(* LS Electric XG5000 project: 201209_AX_ROOF *)
(* PLC NewPLC *)
(* module base 0 slot 0: FEnet:XGL-EFMT(B) (Fast Ethernet 통신 모듈, 전기 Master) *)
(* module base 0 slot 1: FEnet:XGL-EFMT(B) (Fast Ethernet 통신 모듈, 전기 Master) *)
(* module base 0 slot 2: FEnet:XGL-EFMT(B) (Fast Ethernet 통신 모듈, 전기 Master) *)
(* module base 0 slot 3: FEnet:XGL-EFMT(B) (Fast Ethernet 통신 모듈, 전기 Master) *)
(* module base 0 slot 4: FEnet:XGL-EFMT(B) (Fast Ethernet 통신 모듈, 전기 Master) *)
(* module base 0 slot 5: FEnet:XGL-EFMT(B) (Fast Ethernet 통신 모듈, 전기 Master) *)
(* module base 0 slot 6: FEnet:XGL-EFMT(B) (Fast Ethernet 통신 모듈, 전기 Master) *)
(* module base 0 slot 7: FEnet:XGL-EFMT(B) (Fast Ethernet 통신 모듈, 전기 Master) *)
(* module base 0 slot 8: Pnet:XGL-PMEC/B (Pnet 통신 모듈, Profibus-DP Master) *)
(* module base 0 slot 0: 입력 모듈:XBE-DC16A/B (DC24V 입력, 16점 / DC12/24V 입력, 16점) *)
(* module base 0 slot 1: 입력 모듈:XBE-DC16A/B (DC24V 입력, 16점 / DC12/24V 입력, 16점) *)
(* module base 0 slot 2: 입력 모듈:XBE-DC16A/B (DC24V 입력, 16점 / DC12/24V 입력, 16점) *)
(* module base 0 slot 3: 입력 모듈:XBE-DC16A/B (DC24V 입력, 16점 / DC12/24V 입력, 16점) *)
(* module base 0 slot 4: 출력 모듈:XBE-TN/TP16A (트랜지스터 출력, 16점 (싱크출력/소스출력)) *)
(* module base 0 slot 5: 출력 모듈:XBE-TN/TP16A (트랜지스터 출력, 16점 (싱크출력/소스출력)) *)
(* module base 0 slot 6: 출력 모듈:XBE-TN/TP16A (트랜지스터 출력, 16점 (싱크출력/소스출력)) *)
(* module base 0 slot 7: 출력 모듈:XBE-TN/TP16A (트랜지스터 출력, 16점 (싱크출력/소스출력)) *)
(* module base 0 slot 0: 입력 모듈:XBE-DC16A/B (DC24V 입력, 16점 / DC12/24V 입력, 16점) *)
(* module base 0 slot 1: 입력 모듈:XBE-DC16A/B (DC24V 입력, 16점 / DC12/24V 입력, 16점) *)
(* module base 0 slot 2: 입력 모듈:XBE-DC16A/B (DC24V 입력, 16점 / DC12/24V 입력, 16점) *)
(* module base 0 slot 3: 입력 모듈:XBE-DC16A/B (DC24V 입력, 16점 / DC12/24V 입력, 16점) *)
(* module base 0 slot 4: 출력 모듈:XBE-TN/TP16A (트랜지스터 출력, 16점 (싱크출력/소스출력)) *)
(* module base 0 slot 5: 출력 모듈:XBE-TN/TP16A (트랜지스터 출력, 16점 (싱크출력/소스출력)) *)
(* module base 0 slot 6: 출력 모듈:XBE-TN/TP16A (트랜지스터 출력, 16점 (싱크출력/소스출력)) *)
(* module base 0 slot 7: 출력 모듈:XBE-TN/TP16A (트랜지스터 출력, 16점 (싱크출력/소스출력)) *)
(* module base 0 slot 0: 입력 모듈:XBE-DC16A/B (DC24V 입력, 16점 / DC12/24V 입력, 16점) *)
(* module base 0 slot 1: 입력 모듈:XBE-DC16A/B (DC24V 입력, 16점 / DC12/24V 입력, 16점) *)
(* module base 0 slot 2: 입력 모듈:XBE-DC16A/B (DC24V 입력, 16점 / DC12/24V 입력, 16점) *)
(* module base 0 slot 3: 출력 모듈:XBE-TN/TP16A (트랜지스터 출력, 16점 (싱크출력/소스출력)) *)
(* module base 0 slot 4: 출력 모듈:XBE-TN/TP16A (트랜지스터 출력, 16점 (싱크출력/소스출력)) *)
(* module base 0 slot 0: 입력 모듈:XBE-DC16A/B (DC24V 입력, 16점 / DC12/24V 입력, 16점) *)
(* module base 0 slot 1: 입력 모듈:XBE-DC16A/B (DC24V 입력, 16점 / DC12/24V 입력, 16점) *)
(* module base 0 slot 2: 입력 모듈:XBE-DC16A/B (DC24V 입력, 16점 / DC12/24V 입력, 16점) *)
(* module base 0 slot 3: 출력 모듈:XBE-TN/TP16A (트랜지스터 출력, 16점 (싱크출력/소스출력)) *)
(* module base 0 slot 4: 출력 모듈:XBE-TN/TP16A (트랜지스터 출력, 16점 (싱크출력/소스출력)) *)
(* module base 0 slot 0: 입력 모듈:XBE-DC16A/B (DC24V 입력, 16점 / DC12/24V 입력, 16점) *)
(* module base 0 slot 1: 입력 모듈:XBE-DC16A/B (DC24V 입력, 16점 / DC12/24V 입력, 16점) *)
(* module base 0 slot 2: 입력 모듈:XBE-DC16A/B (DC24V 입력, 16점 / DC12/24V 입력, 16점) *)
(* module base 0 slot 3: 출력 모듈:XBE-TN/TP16A (트랜지스터 출력, 16점 (싱크출력/소스출력)) *)
(* module base 0 slot 4: 출력 모듈:XBE-TN/TP16A (트랜지스터 출력, 16점 (싱크출력/소스출력)) *)
(* module base 0 slot 0: 입력 모듈:XBE-DC16A/B (DC24V 입력, 16점 / DC12/24V 입력, 16점) *)
(* module base 0 slot 1: 입력 모듈:XBE-DC16A/B (DC24V 입력, 16점 / DC12/24V 입력, 16점) *)
(* module base 0 slot 2: 입력 모듈:XBE-DC16A/B (DC24V 입력, 16점 / DC12/24V 입력, 16점) *)
(* module base 0 slot 3: 출력 모듈:XBE-TN/TP16A (트랜지스터 출력, 16점 (싱크출력/소스출력)) *)
(* module base 0 slot 4: 출력 모듈:XBE-TN/TP16A (트랜지스터 출력, 16점 (싱크출력/소스출력)) *)
(* module base 0 slot 0: 입력 모듈:XBE-DC16A/B (DC24V 입력, 16점 / DC12/24V 입력, 16점) *)
(* module base 0 slot 1: 입력 모듈:XBE-DC16A/B (DC24V 입력, 16점 / DC12/24V 입력, 16점) *)
(* module base 0 slot 2: 입력 모듈:XBE-DC16A/B (DC24V 입력, 16점 / DC12/24V 입력, 16점) *)
(* module base 0 slot 3: 출력 모듈:XBE-TN/TP16A (트랜지스터 출력, 16점 (싱크출력/소스출력)) *)
(* module base 0 slot 4: 출력 모듈:XBE-TN/TP16A (트랜지스터 출력, 16점 (싱크출력/소스출력)) *)
(* module base 0 slot 0: 입력 모듈:XBE-DC16A/B (DC24V 입력, 16점 / DC12/24V 입력, 16점) *)
(* module base 0 slot 1: 입력 모듈:XBE-DC16A/B (DC24V 입력, 16점 / DC12/24V 입력, 16점) *)
(* module base 0 slot 2: 입력 모듈:XBE-DC16A/B (DC24V 입력, 16점 / DC12/24V 입력, 16점) *)
(* module base 0 slot 3: 출력 모듈:XBE-TN/TP16A (트랜지스터 출력, 16점 (싱크출력/소스출력)) *)
(* module base 0 slot 4: 출력 모듈:XBE-TN/TP16A (트랜지스터 출력, 16점 (싱크출력/소스출력)) *)
(* module base 0 slot 0: 입력 모듈:XBE-DC16A/B (DC24V 입력, 16점 / DC12/24V 입력, 16점) *)
(* module base 0 slot 1: 입력 모듈:XBE-DC16A/B (DC24V 입력, 16점 / DC12/24V 입력, 16점) *)
(* module base 0 slot 2: 입력 모듈:XBE-DC16A/B (DC24V 입력, 16점 / DC12/24V 입력, 16점) *)
(* module base 0 slot 3: 출력 모듈:XBE-TN/TP16A (트랜지스터 출력, 16점 (싱크출력/소스출력)) *)
(* module base 0 slot 4: 출력 모듈:XBE-TN/TP16A (트랜지스터 출력, 16점 (싱크출력/소스출력)) *)
(* module base 0 slot 0: 입력 모듈:XBE-DC16A/B (DC24V 입력, 16점 / DC12/24V 입력, 16점) *)
(* module base 0 slot 1: 입력 모듈:XBE-DC16A/B (DC24V 입력, 16점 / DC12/24V 입력, 16점) *)
(* module base 0 slot 2: 입력 모듈:XBE-DC16A/B (DC24V 입력, 16점 / DC12/24V 입력, 16점) *)
(* module base 0 slot 3: 출력 모듈:XBE-TN/TP16A (트랜지스터 출력, 16점 (싱크출력/소스출력)) *)
(* module base 0 slot 4: 출력 모듈:XBE-TN/TP16A (트랜지스터 출력, 16점 (싱크출력/소스출력)) *)
(* module base 0 slot 0: 입력 모듈:XBE-DC16A/B (DC24V 입력, 16점 / DC12/24V 입력, 16점) *)
(* module base 0 slot 1: 입력 모듈:XBE-DC16A/B (DC24V 입력, 16점 / DC12/24V 입력, 16점) *)
(* module base 0 slot 2: 입력 모듈:XBE-DC16A/B (DC24V 입력, 16점 / DC12/24V 입력, 16점) *)
(* module base 0 slot 3: 출력 모듈:XBE-TN/TP16A (트랜지스터 출력, 16점 (싱크출력/소스출력)) *)
(* module base 0 slot 4: 출력 모듈:XBE-TN/TP16A (트랜지스터 출력, 16점 (싱크출력/소스출력)) *)
(* module base 0 slot 0: 입력 모듈:XBE-DC16A/B (DC24V 입력, 16점 / DC12/24V 입력, 16점) *)
(* module base 0 slot 1: 출력 모듈:XBE-TN/TP16A (트랜지스터 출력, 16점 (싱크출력/소스출력)) *)
(* module base 0 slot 2: 입력 모듈:XBE-DC16A/B (DC24V 입력, 16점 / DC12/24V 입력, 16점) *)
(* module base 0 slot 3: 출력 모듈:XBE-TN/TP16A (트랜지스터 출력, 16점 (싱크출력/소스출력)) *)
(* module base 0 slot 0: 입력 모듈:XBE-DC16A/B (DC24V 입력, 16점 / DC12/24V 입력, 16점) *)
(* module base 0 slot 1: 출력 모듈:XBE-TN/TP16A (트랜지스터 출력, 16점 (싱크출력/소스출력)) *)
(* module base 0 slot 2: 입력 모듈:XBE-DC16A/B (DC24V 입력, 16점 / DC12/24V 입력, 16점) *)
(* module base 0 slot 3: 출력 모듈:XBE-TN/TP16A (트랜지스터 출력, 16점 (싱크출력/소스출력)) *)
(* module base 0 slot 0: 입력 모듈:XBE-DC16A/B (DC24V 입력, 16점 / DC12/24V 입력, 16점) *)
(* module base 0 slot 1: 출력 모듈:XBE-TN/TP16A (트랜지스터 출력, 16점 (싱크출력/소스출력)) *)
(* module base 0 slot 2: 입력 모듈:XBE-DC16A/B (DC24V 입력, 16점 / DC12/24V 입력, 16점) *)
(* module base 0 slot 3: 출력 모듈:XBE-TN/TP16A (트랜지스터 출력, 16점 (싱크출력/소스출력)) *)
(* module base 0 slot 0: 입력 모듈:XBE-DC16A/B (DC24V 입력, 16점 / DC12/24V 입력, 16점) *)
(* module base 0 slot 1: 입력 모듈:XBE-DC16A/B (DC24V 입력, 16점 / DC12/24V 입력, 16점) *)
(* module base 0 slot 2: 입력 모듈:XBE-DC16A/B (DC24V 입력, 16점 / DC12/24V 입력, 16점) *)
(* module base 0 slot 3: 출력 모듈:XBE-TN/TP16A (트랜지스터 출력, 16점 (싱크출력/소스출력)) *)
(* module base 0 slot 4: 출력 모듈:XBE-TN/TP16A (트랜지스터 출력, 16점 (싱크출력/소스출력)) *)
(* module base 0 slot 5: 입력 모듈:XBE-DC16A/B (DC24V 입력, 16점 / DC12/24V 입력, 16점) *)
(* module base 0 slot 6: 출력 모듈:XBE-TN/TP16A (트랜지스터 출력, 16점 (싱크출력/소스출력)) *)
(* module base 0 slot 0: 입력 모듈:XBE-DC16A/B (DC24V 입력, 16점 / DC12/24V 입력, 16점) *)
(* module base 0 slot 1: 출력 모듈:XBE-TN/TP16A (트랜지스터 출력, 16점 (싱크출력/소스출력)) *)
(* module base 0 slot 2: 입력 모듈:XBE-DC16A/B (DC24V 입력, 16점 / DC12/24V 입력, 16점) *)
(* module base 0 slot 3: 출력 모듈:XBE-TN/TP16A (트랜지스터 출력, 16점 (싱크출력/소스출력)) *)
(* module base 0 slot 0: 입력 모듈:XBE-DC16A/B (DC24V 입력, 16점 / DC12/24V 입력, 16점) *)
(* module base 0 slot 1: 출력 모듈:XBE-TN/TP16A (트랜지스터 출력, 16점 (싱크출력/소스출력)) *)
(* module base 0 slot 2: 입력 모듈:XBE-DC16A/B (DC24V 입력, 16점 / DC12/24V 입력, 16점) *)
(* module base 0 slot 3: 출력 모듈:XBE-TN/TP16A (트랜지스터 출력, 16점 (싱크출력/소스출력)) *)
(* module base 0 slot 0: 입력 모듈:XBE-DC16A/B (DC24V 입력, 16점 / DC12/24V 입력, 16점) *)
(* module base 0 slot 1: 입력 모듈:XBE-DC16A/B (DC24V 입력, 16점 / DC12/24V 입력, 16점) *)
(* module base 0 slot 2: 입력 모듈:XBE-DC16A/B (DC24V 입력, 16점 / DC12/24V 입력, 16점) *)
(* module base 0 slot 3: 출력 모듈:XBE-TN/TP16A (트랜지스터 출력, 16점 (싱크출력/소스출력)) *)
(* module base 0 slot 4: 출력 모듈:XBE-TN/TP16A (트랜지스터 출력, 16점 (싱크출력/소스출력)) *)
(* module base 0 slot 5: 입력 모듈:XBE-DC16A/B (DC24V 입력, 16점 / DC12/24V 입력, 16점) *)
(* module base 0 slot 6: 출력 모듈:XBE-TN/TP16A (트랜지스터 출력, 16점 (싱크출력/소스출력)) *)
(* module base 0 slot 0: 입력 모듈:XBE-DC16A/B (DC24V 입력, 16점 / DC12/24V 입력, 16점) *)
(* module base 0 slot 1: 입력 모듈:XBE-DC16A/B (DC24V 입력, 16점 / DC12/24V 입력, 16점) *)
(* module base 0 slot 2: 입력 모듈:XBE-DC16A/B (DC24V 입력, 16점 / DC12/24V 입력, 16점) *)
(* module base 0 slot 3: 출력 모듈:XBE-TN/TP16A (트랜지스터 출력, 16점 (싱크출력/소스출력)) *)
(* module base 0 slot 4: 출력 모듈:XBE-TN/TP16A (트랜지스터 출력, 16점 (싱크출력/소스출력)) *)
(* module base 0 slot 5: 입력 모듈:XBE-DC16A/B (DC24V 입력, 16점 / DC12/24V 입력, 16점) *)
(* module base 0 slot 6: 출력 모듈:XBE-TN/TP16A (트랜지스터 출력, 16점 (싱크출력/소스출력)) *)
(* module base 0 slot 0: 입력 모듈:XBE-DC16A/B (DC24V 입력, 16점 / DC12/24V 입력, 16점) *)
(* module base 0 slot 1: 입력 모듈:XBE-DC16A/B (DC24V 입력, 16점 / DC12/24V 입력, 16점) *)
(* module base 0 slot 2: 출력 모듈:XBE-TN/TP16A (트랜지스터 출력, 16점 (싱크출력/소스출력)) *)
(* module base 0 slot 3: 입력 모듈:XBE-DC16A/B (DC24V 입력, 16점 / DC12/24V 입력, 16점) *)
(* module base 0 slot 4: 출력 모듈:XBE-TN/TP16A (트랜지스터 출력, 16점 (싱크출력/소스출력)) *)
(* module base 0 slot 0: 입력 모듈:XBE-DC16A/B (DC24V 입력, 16점 / DC12/24V 입력, 16점) *)
(* module base 0 slot 1: 입력 모듈:XBE-DC16A/B (DC24V 입력, 16점 / DC12/24V 입력, 16점) *)
(* module base 0 slot 2: 출력 모듈:XBE-TN/TP16A (트랜지스터 출력, 16점 (싱크출력/소스출력)) *)
(* module base 0 slot 3: 입력 모듈:XBE-DC16A/B (DC24V 입력, 16점 / DC12/24V 입력, 16점) *)
(* module base 0 slot 4: 출력 모듈:XBE-TN/TP16A (트랜지스터 출력, 16점 (싱크출력/소스출력)) *)
(* module base 0 slot 0: 입력 모듈:XBE-DC16A/B (DC24V 입력, 16점 / DC12/24V 입력, 16점) *)
(* module base 0 slot 1: 입력 모듈:XBE-DC16A/B (DC24V 입력, 16점 / DC12/24V 입력, 16점) *)
(* module base 0 slot 2: 출력 모듈:XBE-TN/TP16A (트랜지스터 출력, 16점 (싱크출력/소스출력)) *)
(* module base 0 slot 3: 입력 모듈:XBE-DC16A/B (DC24V 입력, 16점 / DC12/24V 입력, 16점) *)
(* module base 0 slot 4: 출력 모듈:XBE-TN/TP16A (트랜지스터 출력, 16점 (싱크출력/소스출력)) *)
(* module base 0 slot 0: 입력 모듈:XBE-DC16A/B (DC24V 입력, 16점 / DC12/24V 입력, 16점) *)
(* module base 0 slot 1: 입력 모듈:XBE-DC16A/B (DC24V 입력, 16점 / DC12/24V 입력, 16점) *)
(* module base 0 slot 2: 입력 모듈:XBE-DC16A/B (DC24V 입력, 16점 / DC12/24V 입력, 16점) *)
(* module base 0 slot 3: 출력 모듈:XBE-TN/TP16A (트랜지스터 출력, 16점 (싱크출력/소스출력)) *)
(* module base 0 slot 4: 출력 모듈:XBE-TN/TP16A (트랜지스터 출력, 16점 (싱크출력/소스출력)) *)
(* module base 0 slot 5: 입력 모듈:XBE-DC16A/B (DC24V 입력, 16점 / DC12/24V 입력, 16점) *)
(* module base 0 slot 6: 출력 모듈:XBE-TN/TP16A (트랜지스터 출력, 16점 (싱크출력/소스출력)) *)
VAR_GLOBAL RETAIN
    ALWAYS_OFF AT %MW3.0 : BOOL; (* 항시 OFF *)
    ALWAYS_ON AT %MW3.1 : BOOL; (* 항시 ON *)
    CARTYPE AT %MW10000 : ARRAY[0..599] OF WORD; (* CARTYPE *)
    CLOCK_BIT_0_1Sec AT %MW0.0 : BOOL; (* CLOCK_BIT_0_1Sec *)
    CLOCK_BIT_0_2Sec AT %MW0.1 : BOOL; (* CLOCK_BIT_0_2Sec *)
    CLOCK_BIT_0_4Sec AT %MW0.2 : BOOL; (* CLOCK_BIT_0_4Sec *)
    CLOCK_BIT_0_5Sec AT %MW0.3 : BOOL; (* 플리커 0.5초 *)
    CLOCK_BIT_0_8Sec AT %MW0.4 : BOOL; (* CLOCK_BIT_0_8Sec *)
    CLOCK_BIT_1_0Sec AT %MW0.5 : BOOL; (* CLOCK_BIT_1_0Sec *)
    CLOCK_BIT_1_6Sec AT %MW0.6 : BOOL; (* CLOCK_BIT_1_6Sec *)
    CLOCK_BIT_2_0Sec AT %MW0.7 : BOOL; (* CLOCK_BIT_2_0Sec *)
    GATE1_M_CP_TRIP AT %MW400.15 : BOOL; (* GATEBOX1 CP OFF 이상 *)
    GATE1_M_EMSTOP AT %MW400.7 : BOOL; (* GATE1 비상정지 이상 *)
    GATE1_M_GATE_CLOSE AT %MW400.3 : BOOL; (* GATE1_M_GATE_CLOSE *)
    GATE1_M_GATE_OPEN AT %MW400.13 : BOOL; (* GATEBOX1 이상 *)
    GATE1_M_GATE_열림_보조 AT %MW400.12 : BOOL; (* GATE1_M_GATE_열림_보조 *)
    GATE1_M_RESTART AT %MW400.1 : BOOL; (* GATE1_M_RESTART *)
    GATE1_M_STOP_CALL AT %MW400.2 : BOOL; (* GATE1_M_STOP_CALL *)
    GATE1_M_비상정지_정상 AT %MW400.4 : BOOL;
    GATE1_M_이상_리셋 AT %MW400.0 : BOOL; (* GATE1 PB 이상리셋 *)
    GATE1_M_통신_이상 AT %MW400.14 : BOOL; (* GATEBOX1 통신이상 *)
    GATE2_M_CP_TRIP AT %MW401.15 : BOOL; (* GATEBOX2 CP OFF 이상 *)
    GATE2_M_EMSTOP AT %MW401.7 : BOOL; (* GATE2 비상정지 이상 *)
    GATE2_M_GATE_CLOSE AT %MW401.3 : BOOL; (* GATE2_M_GATE_CLOSE *)
    GATE2_M_GATE_OPEN AT %MW401.13 : BOOL; (* GATEBOX2 이상 *)
    GATE2_M_GATE_열림_보조 AT %MW401.12 : BOOL; (* GATE2_M_GATE_열림_보조 *)
    GATE2_M_RESTART AT %MW401.1 : BOOL; (* GATE2_M_RESTART *)
    GATE2_M_STOP_CALL AT %MW401.2 : BOOL; (* GATE2_M_STOP_CALL *)
    GATE2_M_비상정지_정상 AT %MW401.4 : BOOL;
    GATE2_M_이상_리셋 AT %MW401.0 : BOOL; (* GATE2 PB 이상리셋 *)
    GATE2_M_통신_이상 AT %MW401.14 : BOOL; (* GATEBOX2 통신이상 *)
    GATE3_M_CP_TRIP AT %MW402.15 : BOOL; (* GATEBOX3 CP OFF 이상 *)
    GATE3_M_EMSTOP AT %MW402.7 : BOOL; (* GATE3 비상정지 이상 *)
    GATE3_M_GATE_CLOSE AT %MW402.3 : BOOL; (* GATE3_M_GATE_CLOSE *)
    GATE3_M_GATE_OPEN AT %MW402.13 : BOOL; (* GATEBOX3 이상 *)
    GATE3_M_GATE_열림_보조 AT %MW402.12 : BOOL; (* GATE3_M_GATE_열림_보조 *)
    GATE3_M_RESTART AT %MW402.1 : BOOL; (* GATE3_M_RESTART *)
    GATE3_M_STOP_CALL AT %MW402.2 : BOOL; (* GATE3_M_STOP_CALL *)
    GATE3_M_비상정지_정상 AT %MW402.4 : BOOL;
    GATE3_M_이상_리셋 AT %MW402.0 : BOOL; (* GATE3 PB 이상리셋 *)
    GATE3_M_통신_이상 AT %MW402.14 : BOOL; (* GATEBOX3 통신이상 *)
    GATE4_M_CP_TRIP AT %MW403.15 : BOOL;
    GATE4_M_EMSTOP AT %MW403.7 : BOOL;
    GATE4_M_GATE_CLOSE AT %MW403.3 : BOOL;
    GATE4_M_GATE_OPEN AT %MW403.13 : BOOL;
    GATE4_M_GATE_열림_보조 AT %MW403.12 : BOOL;
    GATE4_M_RESTART AT %MW403.1 : BOOL;
    GATE4_M_STOP_CALL AT %MW403.2 : BOOL;
    GATE4_M_비상정지_정상 AT %MW403.4 : BOOL;
    GATE4_M_이상_리셋 AT %MW403.0 : BOOL;
    GATE4_M_통신_이상 AT %MW403.14 : BOOL;
    GATE5_M_CP_TRIP AT %MW404.15 : BOOL;
    GATE5_M_EMSTOP AT %MW404.7 : BOOL;
    GATE5_M_GATE_CLOSE AT %MW404.3 : BOOL;
    GATE5_M_GATE_OPEN AT %MW404.13 : BOOL;
    GATE5_M_GATE_열림_보조 AT %MW404.12 : BOOL;
    GATE5_M_RESTART AT %MW404.1 : BOOL;
    GATE5_M_STOP_CALL AT %MW404.2 : BOOL;
    GATE5_M_비상정지_정상 AT %MW404.4 : BOOL;
    GATE5_M_이상_리셋 AT %MW404.0 : BOOL;
    GATE5_M_통신_이상 AT %MW404.14 : BOOL;
    HMI_M_매칭_R361_1_S366 AT %MW70.0 : BOOL;
    HMI_M_매칭_S366_R361_1 AT %MW70.1 : BOOL;
    HMI_M_매칭선택 AT %MW70 : WORD;
    HMI_M_매칭차종_DATA_OK AT %MW9.9 : BOOL;
    HMI_M_매칭차종_복사_ON AT %MW9.6 : BOOL;
    HMI_M_매칭차종_복사_SET AT %MW9.8 : BOOL;
    HMI_M_매칭차종_복사_가능 AT %MW9.7 : BOOL;
    HMI_M_선택_MOD_CARR AT %MW12 : WORD;
    HMI_M_선택_MOD_PROF AT %MW13 : WORD;
    HMI_M_선택_MOD_ROOF_RACK AT %MW6.1 : BOOL; (* HMI M 선택 MOD S363 *)
    HMI_M_선택_MOD_S362 AT %MW6.0 : BOOL; (* HMI M 선택 MOD S362 *)
    HMI_M_선택_MOD_S364 AT %MW6.2 : BOOL; (* HMI M 선택 MOD S364 *)
    HMI_M_선택_MOD_S365 AT %MW6.3 : BOOL; (* HMI M 선택 MOD S365 *)
    HMI_M_선택_MOD_S366 AT %MW6.4 : BOOL; (* HMI M 선택 MOD S366 *)
    HMI_M_선택_MOD_S367 AT %MW6.5 : BOOL; (* HMI M 선택 MOD S367 *)
    HMI_M_선택_MOD_S368 AT %MW6.6 : BOOL; (* HMI M 선택 MOD S368 *)
    HMI_M_선택_MOD_S369_1 AT %MW6.7 : BOOL; (* HMI M 선택 MOD S369_1 *)
    HMI_M_선택_MOD_S369_LD AT %MW6.8 : BOOL; (* HMI M 선택 MOD S369 *)
    HMI_M_선택_MOD_S369_UD AT %MW6.9 : BOOL;
    HMI_M_선택_MOD_STN AT %MW6 : WORD; (* HMI M 선택 MOD STN *)
    HMI_M_차종매칭 AT %MW50 : ARRAY[0..19] OF WORD;
    HMI_M_차종매칭_SEQ AT %MW50 : WORD;
    HMI_M_차종매칭_VIN_NO_1_2 AT %MW61 : WORD;
    HMI_M_차종매칭_VIN_NO_3_4 AT %MW62 : WORD;
    HMI_M_차종매칭_VIN_NO_5_6 AT %MW63 : WORD;
    HMI_M_차종매칭_VIN_NO_7_8 AT %MW64 : WORD;
    HMI_M_차종매칭_VIN_NO_9_10 AT %MW65 : WORD;
    HMI_M_차종매칭_차종1_AX AT %MW51.0 : BOOL;
    HMI_M_차종매칭_차종1_B AT %MW51.1 : BOOL;
    HMI_M_차종매칭_차종1_C AT %MW51.2 : BOOL;
    HMI_M_차종매칭_차종1_D AT %MW51.3 : BOOL;
    HMI_M_차종매칭_차종1_E AT %MW51.4 : BOOL;
    HMI_M_차종매칭_차종1_F AT %MW51.5 : BOOL;
    HMI_M_차종매칭_차종1_G AT %MW51.6 : BOOL;
    HMI_M_차종매칭_차종1_H AT %MW51.7 : BOOL;
    HMI_M_차종매칭_차종2_3DR AT %MW51.8 : BOOL;
    HMI_M_차종매칭_차종2_4DR AT %MW51.9 : BOOL;
    HMI_M_차종매칭_차종2_5DR AT %MW51.10 : BOOL;
    HMI_M_차종매칭_차종2_SP1 AT %MW51.12 : BOOL;
    HMI_M_차종매칭_차종2_SP2 AT %MW51.13 : BOOL;
    HMI_M_차종매칭_차종2_WGN AT %MW51.11 : BOOL;
    HMI_M_차종매칭_차종3_LHD AT %MW51.14 : BOOL;
    HMI_M_차종매칭_차종3_RHD AT %MW51.15 : BOOL;
    HMI_M_차종매칭_차종4_EEC AT %MW52.3 : BOOL;
    HMI_M_차종매칭_차종4_SP1 AT %MW52.8 : BOOL;
    HMI_M_차종매칭_차종4_SP2 AT %MW52.9 : BOOL;
    HMI_M_차종매칭_차종4_SP3 AT %MW52.11 : BOOL;
    HMI_M_차종매칭_차종4_SP4 AT %MW52.12 : BOOL;
    HMI_M_차종매칭_차종4_SP5 AT %MW52.13 : BOOL;
    HMI_M_차종매칭_차종4_SP6 AT %MW52.14 : BOOL;
    HMI_M_차종매칭_차종4_SP7 AT %MW52.15 : BOOL;
    HMI_M_차종매칭_차종4_내수 AT %MW52.0 : BOOL;
    HMI_M_차종매칭_차종4_러시아 AT %MW52.10 : BOOL;
    HMI_M_차종매칭_차종4_북미 AT %MW52.2 : BOOL;
    HMI_M_차종매칭_차종4_브라질 AT %MW52.7 : BOOL;
    HMI_M_차종매칭_차종4_수출 AT %MW52.1 : BOOL;
    HMI_M_차종매칭_차종4_중국 AT %MW52.6 : BOOL;
    HMI_M_차종매칭_차종4_중동 AT %MW52.5 : BOOL;
    HMI_M_차종매칭_차종4_호주 AT %MW52.4 : BOOL;
    HMI_M_차종매칭_차종5_AT AT %MW53.1 : BOOL;
    HMI_M_차종매칭_차종5_MT AT %MW53.0 : BOOL;
    HMI_M_차종매칭_차종5_SP1 AT %MW53.2 : BOOL;
    HMI_M_차종매칭_차종6_DSROOF AT %MW53.6 : BOOL;
    HMI_M_차종매칭_차종6_SP1 AT %MW53.7 : BOOL;
    HMI_M_차종매칭_차종6_썬루프 AT %MW53.4 : BOOL;
    HMI_M_차종매칭_차종6_일반루프 AT %MW53.3 : BOOL;
    HMI_M_차종매칭_차종6_파노라마루프 AT %MW53.5 : BOOL;
    HMI_M_차종매칭_차종7_DSL AT %MW53.9 : BOOL;
    HMI_M_차종매칭_차종7_GSL AT %MW53.8 : BOOL;
    HMI_M_차종매칭_차종7_SP1 AT %MW53.10 : BOOL;
    HMI_M_차종매칭_차종7_SP2 AT %MW53.11 : BOOL;
    HMI_M_차종매칭_차종7_SP3 AT %MW53.12 : BOOL;
    HMI_M_차종매칭_차종7_SP4 AT %MW53.13 : BOOL;
    HMI_M_차종매칭_차종7_SP5 AT %MW53.14 : BOOL;
    HMI_M_차종매칭_차종7_SP6 AT %MW53.15 : BOOL;
    HMI_M_차종매칭_차종8_2WD AT %MW54.0 : BOOL;
    HMI_M_차종매칭_차종8_4WD AT %MW54.1 : BOOL;
    HMI_M_차종매칭_차종8_SP1 AT %MW54.2 : BOOL;
    HMI_M_차종매칭_차종9_MPI AT %MW54.3 : BOOL;
    HMI_M_차종매칭_차종9_SP1 AT %MW54.5 : BOOL;
    HMI_M_차종매칭_차종9_SP10 AT %MW54.14 : BOOL;
    HMI_M_차종매칭_차종9_SP11 AT %MW54.15 : BOOL;
    HMI_M_차종매칭_차종9_SP2 AT %MW54.6 : BOOL;
    HMI_M_차종매칭_차종9_SP3 AT %MW54.7 : BOOL;
    HMI_M_차종매칭_차종9_SP4 AT %MW54.8 : BOOL;
    HMI_M_차종매칭_차종9_SP5 AT %MW54.9 : BOOL;
    HMI_M_차종매칭_차종9_SP6 AT %MW54.10 : BOOL;
    HMI_M_차종매칭_차종9_SP7 AT %MW54.11 : BOOL;
    HMI_M_차종매칭_차종9_SP8 AT %MW54.12 : BOOL;
    HMI_M_차종매칭_차종9_SP9 AT %MW54.13 : BOOL;
    HMI_M_차종매칭_차종9_T_GDI AT %MW54.4 : BOOL;
    HMI_M_차종매칭_차종_AS AT %MW60.9 : BOOL;
    HMI_M_차종매칭_차종_OPT1_R_RACK_무 AT %MW55.3 : BOOL;
    HMI_M_차종매칭_차종_OPT1_R_RACK_유 AT %MW55.2 : BOOL;
    HMI_M_차종매칭_차종_OPT1_SP1 AT %MW55.10 : BOOL;
    HMI_M_차종매칭_차종_OPT1_SP2 AT %MW55.11 : BOOL;
    HMI_M_차종매칭_차종_OPT1_SP3 AT %MW55.12 : BOOL;
    HMI_M_차종매칭_차종_OPT1_SP4 AT %MW55.13 : BOOL;
    HMI_M_차종매칭_차종_OPT1_SP5 AT %MW55.14 : BOOL;
    HMI_M_차종매칭_차종_OPT1_SP6 AT %MW55.15 : BOOL;
    HMI_M_차종매칭_차종_OPT1_S_REP_EATER_무 AT %MW55.7 : BOOL;
    HMI_M_차종매칭_차종_OPT1_S_REP_EATER_유 AT %MW55.6 : BOOL;
    HMI_M_차종매칭_차종_OPT1_VAN_무 AT %MW55.9 : BOOL;
    HMI_M_차종매칭_차종_OPT1_VAN_유 AT %MW55.8 : BOOL;
    HMI_M_차종매칭_차종_OPT1_슬라이딩_무 AT %MW55.1 : BOOL;
    HMI_M_차종매칭_차종_OPT1_슬라이딩_유 AT %MW55.0 : BOOL;
    HMI_M_차종매칭_차종_OPT1_폴딩_무 AT %MW55.5 : BOOL;
    HMI_M_차종매칭_차종_OPT1_폴딩_유 AT %MW55.4 : BOOL;
    HMI_M_차종매칭_차종_OPT2_SP_WORD1 AT %MW56 : WORD;
    HMI_M_차종매칭_차종_OPT3_SP_WORD2 AT %MW57 : WORD;
    HMI_M_차종매칭_차종_OPT4_SP_WORD3 AT %MW58 : WORD;
    HMI_M_차종매칭_차종_OPT5_SP_WORD4 AT %MW59 : WORD;
    HMI_M_차종매칭_차종_SP1 AT %MW60.0 : BOOL;
    HMI_M_차종매칭_차종_SP2 AT %MW60.1 : BOOL;
    HMI_M_차종매칭_차종_SP3 AT %MW60.2 : BOOL;
    HMI_M_차종매칭_차종_SP4 AT %MW60.3 : BOOL;
    HMI_M_차종매칭_차종_SP5 AT %MW60.4 : BOOL;
    HMI_M_차종매칭_차종_SP6 AT %MW60.5 : BOOL;
    HMI_M_차종매칭_차종_SP7 AT %MW60.6 : BOOL;
    HMI_M_차종매칭_차종_SP8 AT %MW60.7 : BOOL;
    HMI_M_차종매칭_차종_SP9 AT %MW60.15 : BOOL;
    HMI_M_차종매칭_차종_공대차 AT %MW60.12 : BOOL;
    HMI_M_차종매칭_차종_공차 AT %MW60.10 : BOOL;
    HMI_M_차종매칭_차종_불량대차 AT %MW60.13 : BOOL;
    HMI_M_차종매칭_차종_불량차 AT %MW60.11 : BOOL;
    HMI_M_차종매칭_차종_비축 AT %MW60.8 : BOOL;
    HMI_M_차종매칭_차종_취출대차 AT %MW60.14 : BOOL;
    HMI_M_차종수정 AT %MW10 : ARRAY[0..19] OF WORD;
    HMI_M_차종수정_DATA_OK AT %MW9.0 : BOOL;
    HMI_M_차종수정_RESET AT %MW9.2 : BOOL;
    HMI_M_차종수정_SEQ AT %MW10 : WORD;
    HMI_M_차종수정_SET AT %MW9.1 : BOOL;
    HMI_M_차종수정_VIN_NO_1_2 AT %MW21 : WORD;
    HMI_M_차종수정_VIN_NO_3_4 AT %MW22 : WORD;
    HMI_M_차종수정_VIN_NO_5_6 AT %MW23 : WORD;
    HMI_M_차종수정_VIN_NO_7_8 AT %MW24 : WORD;
    HMI_M_차종수정_VIN_NO_9_10 AT %MW25 : WORD;
    HMI_M_차종수정_차종1_AX AT %MW11.0 : BOOL;
    HMI_M_차종수정_차종1_B AT %MW11.1 : BOOL;
    HMI_M_차종수정_차종1_C AT %MW11.2 : BOOL;
    HMI_M_차종수정_차종1_D AT %MW11.3 : BOOL;
    HMI_M_차종수정_차종1_E AT %MW11.4 : BOOL;
    HMI_M_차종수정_차종1_F AT %MW11.5 : BOOL;
    HMI_M_차종수정_차종1_G AT %MW11.6 : BOOL;
    HMI_M_차종수정_차종1_H AT %MW11.7 : BOOL;
    HMI_M_차종수정_차종2_3DR AT %MW11.8 : BOOL;
    HMI_M_차종수정_차종2_4DR AT %MW11.9 : BOOL;
    HMI_M_차종수정_차종2_5DR AT %MW11.10 : BOOL;
    HMI_M_차종수정_차종2_SP1 AT %MW11.12 : BOOL;
    HMI_M_차종수정_차종2_SP2 AT %MW11.13 : BOOL;
    HMI_M_차종수정_차종2_WGN AT %MW11.11 : BOOL;
    HMI_M_차종수정_차종3_LHD AT %MW11.14 : BOOL;
    HMI_M_차종수정_차종3_RHD AT %MW11.15 : BOOL;
    HMI_M_차종수정_차종4_EEC AT %MW12.3 : BOOL;
    HMI_M_차종수정_차종4_SP1 AT %MW12.8 : BOOL;
    HMI_M_차종수정_차종4_SP2 AT %MW12.9 : BOOL;
    HMI_M_차종수정_차종4_SP3 AT %MW12.11 : BOOL;
    HMI_M_차종수정_차종4_SP4 AT %MW12.12 : BOOL;
    HMI_M_차종수정_차종4_SP5 AT %MW12.13 : BOOL;
    HMI_M_차종수정_차종4_SP6 AT %MW12.14 : BOOL;
    HMI_M_차종수정_차종4_SP7 AT %MW12.15 : BOOL;
    HMI_M_차종수정_차종4_내수 AT %MW12.0 : BOOL;
    HMI_M_차종수정_차종4_러시아 AT %MW12.10 : BOOL;
    HMI_M_차종수정_차종4_북미 AT %MW12.2 : BOOL;
    HMI_M_차종수정_차종4_브라질 AT %MW12.7 : BOOL;
    HMI_M_차종수정_차종4_수출 AT %MW12.1 : BOOL;
    HMI_M_차종수정_차종4_중국 AT %MW12.6 : BOOL;
    HMI_M_차종수정_차종4_중동 AT %MW12.5 : BOOL;
    HMI_M_차종수정_차종4_호주 AT %MW12.4 : BOOL;
    HMI_M_차종수정_차종5_AT AT %MW13.1 : BOOL;
    HMI_M_차종수정_차종5_MT AT %MW13.0 : BOOL;
    HMI_M_차종수정_차종5_SP1 AT %MW13.2 : BOOL;
    HMI_M_차종수정_차종6_DSROOF AT %MW13.6 : BOOL;
    HMI_M_차종수정_차종6_SP1 AT %MW13.7 : BOOL;
    HMI_M_차종수정_차종6_썬루프 AT %MW13.4 : BOOL;
    HMI_M_차종수정_차종6_일반루프 AT %MW13.3 : BOOL;
    HMI_M_차종수정_차종6_파노라마루프 AT %MW13.5 : BOOL;
    HMI_M_차종수정_차종7_DSL AT %MW13.9 : BOOL;
    HMI_M_차종수정_차종7_GSL AT %MW13.8 : BOOL;
    HMI_M_차종수정_차종7_SP1 AT %MW13.10 : BOOL;
    HMI_M_차종수정_차종7_SP2 AT %MW13.11 : BOOL;
    HMI_M_차종수정_차종7_SP3 AT %MW13.12 : BOOL;
    HMI_M_차종수정_차종7_SP4 AT %MW13.13 : BOOL;
    HMI_M_차종수정_차종7_SP5 AT %MW13.14 : BOOL;
    HMI_M_차종수정_차종7_SP6 AT %MW13.15 : BOOL;
    HMI_M_차종수정_차종8_2WD AT %MW14.0 : BOOL;
    HMI_M_차종수정_차종8_4WD AT %MW14.1 : BOOL;
    HMI_M_차종수정_차종8_SP1 AT %MW14.2 : BOOL;
    HMI_M_차종수정_차종9_MPI AT %MW14.3 : BOOL;
    HMI_M_차종수정_차종9_SP1 AT %MW14.5 : BOOL;
    HMI_M_차종수정_차종9_SP10 AT %MW14.14 : BOOL;
    HMI_M_차종수정_차종9_SP11 AT %MW14.15 : BOOL;
    HMI_M_차종수정_차종9_SP2 AT %MW14.6 : BOOL;
    HMI_M_차종수정_차종9_SP3 AT %MW14.7 : BOOL;
    HMI_M_차종수정_차종9_SP4 AT %MW14.8 : BOOL;
    HMI_M_차종수정_차종9_SP5 AT %MW14.9 : BOOL;
    HMI_M_차종수정_차종9_SP6 AT %MW14.10 : BOOL;
    HMI_M_차종수정_차종9_SP7 AT %MW14.11 : BOOL;
    HMI_M_차종수정_차종9_SP8 AT %MW14.12 : BOOL;
    HMI_M_차종수정_차종9_SP9 AT %MW14.13 : BOOL;
    HMI_M_차종수정_차종9_T_GDI AT %MW14.4 : BOOL;
    HMI_M_차종수정_차종_AS AT %MW20.9 : BOOL;
    HMI_M_차종수정_차종_OPT1_R_RACK_무 AT %MW15.3 : BOOL;
    HMI_M_차종수정_차종_OPT1_R_RACK_유 AT %MW15.2 : BOOL;
    HMI_M_차종수정_차종_OPT1_SP1 AT %MW15.10 : BOOL;
    HMI_M_차종수정_차종_OPT1_SP2 AT %MW15.11 : BOOL;
    HMI_M_차종수정_차종_OPT1_SP3 AT %MW15.12 : BOOL;
    HMI_M_차종수정_차종_OPT1_SP4 AT %MW15.13 : BOOL;
    HMI_M_차종수정_차종_OPT1_SP5 AT %MW15.14 : BOOL;
    HMI_M_차종수정_차종_OPT1_SP6 AT %MW15.15 : BOOL;
    HMI_M_차종수정_차종_OPT1_S_REP_EATER_무 AT %MW15.7 : BOOL;
    HMI_M_차종수정_차종_OPT1_S_REP_EATER_유 AT %MW15.6 : BOOL;
    HMI_M_차종수정_차종_OPT1_VAN_무 AT %MW15.9 : BOOL;
    HMI_M_차종수정_차종_OPT1_VAN_유 AT %MW15.8 : BOOL;
    HMI_M_차종수정_차종_OPT1_슬라이딩_무 AT %MW15.1 : BOOL;
    HMI_M_차종수정_차종_OPT1_슬라이딩_유 AT %MW15.0 : BOOL;
    HMI_M_차종수정_차종_OPT1_폴딩_무 AT %MW15.5 : BOOL;
    HMI_M_차종수정_차종_OPT1_폴딩_유 AT %MW15.4 : BOOL;
    HMI_M_차종수정_차종_OPT2_SP_WORD1 AT %MW16 : WORD;
    HMI_M_차종수정_차종_OPT3_SP_WORD2 AT %MW17 : WORD;
    HMI_M_차종수정_차종_OPT4_SP_WORD3 AT %MW18 : ARRAY[0..19] OF WORD;
    HMI_M_차종수정_차종_OPT5_SP_WORD4 AT %MW19 : WORD;
    HMI_M_차종수정_차종_SP1 AT %MW20.0 : BOOL;
    HMI_M_차종수정_차종_SP2 AT %MW20.1 : BOOL;
    HMI_M_차종수정_차종_SP3 AT %MW20.2 : BOOL;
    HMI_M_차종수정_차종_SP4 AT %MW20.3 : BOOL;
    HMI_M_차종수정_차종_SP5 AT %MW20.4 : BOOL;
    HMI_M_차종수정_차종_SP6 AT %MW20.5 : BOOL;
    HMI_M_차종수정_차종_SP7 AT %MW20.6 : BOOL;
    HMI_M_차종수정_차종_SP8 AT %MW20.7 : BOOL;
    HMI_M_차종수정_차종_SP9 AT %MW20.15 : BOOL;
    HMI_M_차종수정_차종_공대차 AT %MW20.12 : BOOL;
    HMI_M_차종수정_차종_공차 AT %MW20.10 : BOOL;
    HMI_M_차종수정_차종_불량대차 AT %MW20.13 : BOOL;
    HMI_M_차종수정_차종_불량차 AT %MW20.11 : BOOL;
    HMI_M_차종수정_차종_비축 AT %MW20.8 : BOOL;
    HMI_M_차종수정_차종_취출대차 AT %MW20.14 : BOOL;
    HMI_M_차종수정가능_OK AT %MW9.4 : BOOL;
    HMI_M_차종수정가능_SEL AT %MW9.3 : BOOL;
    HMI_M_현재표출_차종 AT %MW30 : ARRAY[0..19] OF WORD;
    HMI_차종매칭_공정선택 AT %MW8 : WORD;
    HMI_차종수정_공정선택 AT %MW7 : WORD;
    HOP1_M_CP_OFF_이상 AT %MW360.15 : BOOL; (* HOP1 CP OFF 이상 *)
    HOP1_M_EM_STOP_정상 AT %MW360.8 : BOOL;
    HOP1_M_램프_테스트 AT %MW360.6 : BOOL; (* HOP1_M_램프_테스트 *)
    HOP1_M_부저_정지 AT %MW360.5 : BOOL; (* HOP1 PB 부저정지 *)
    HOP1_M_비상정지 AT %MW360.7 : BOOL; (* HOP1 비상정지 이상 *)
    HOP1_M_수동모드 AT %MW360.1 : BOOL; (* HOP1_M_수동모드 *)
    HOP1_M_운전준비_ON AT %MW360.0 : BOOL; (* HOP1_M_운전준비_ON *)
    HOP1_M_이상_리셋 AT %MW360.4 : BOOL; (* HOP1 PB 이상리셋 *)
    HOP1_M_자동_START AT %MW360.3 : BOOL; (* HOP1_M_자동_START *)
    HOP1_M_자동모드 AT %MW360.2 : BOOL; (* HOP1_M_자동모드 *)
    HOP1_M_통신_이상 AT %MW360.14 : BOOL; (* HOP1 통신이상 *)
    INV1_M_CP_OFF_이상 AT %MW355.3 : BOOL; (* 인버터반1 CP OFF 이상 *)
    INV1_M_PS_DC_LOW AT %MW355.2 : BOOL; (* 인버터반1 PS저전압 이상 *)
    INV1_M_SPD_이상 AT %MW355.1 : BOOL; (* 인버터반1 SPD 이상 *)
    INV1_M_총괄_이상 AT %MW355.0 : BOOL; (* INV1_M_총괄_이상 *)
    INV1_M_통신_이상 AT %MW355.4 : BOOL; (* 인버터반1 통신이상 *)
    MCP_M_CP_OFF_이상 AT %MW351.0 : BOOL; (* MCP CP OFF 이상총괄 *)
    MCP_M_DISPLAY_CP_TRIP AT %MW351.6 : BOOL; (* MCP 출력전원 CP OFF 이상 *)
    MCP_M_HUB_CP_TRIP AT %MW351.1 : BOOL; (* MCP PS전원 CP OFF 이상 *)
    MCP_M_INPUT_CP_TRIP AT %MW351.3 : BOOL; (* MCP HUB전원  CP OFF 이상 *)
    MCP_M_OUTPUT_CP_TRIP AT %MW351.4 : BOOL; (* MCP 통신모듈 전원 CP OFF 이상 *)
    MCP_M_OUTPUT_MC_OFF AT %MW350.11 : BOOL; (* MCP_M_OUTPUT_MC_OFF *)
    MCP_M_OUTPUT_MC_ON AT %MW350.10 : BOOL; (* MCP_M_OUTPUT_MC_ON *)
    MCP_M_OUTPUT_MC_이상 AT %MW354.8 : BOOL; (* MCP 운전준비 MC 이상 *)
    MCP_M_PROFI_PWR_CP_TRIP AT %MW351.5 : BOOL; (* MCP 입력전원 CP OFF 이상 *)
    MCP_M_PS1_DC_LOW AT %MW353.1 : BOOL; (* MCP PS1 전원 이상 *)
    MCP_M_PS2_DC_LOW AT %MW353.2 : BOOL; (* MCP PS2 전원 이상 *)
    MCP_M_PS3_DC_LOW AT %MW353.3 : BOOL; (* MCP PS3 전원 이상 *)
    MCP_M_PS4_DC_LOW AT %MW353.4 : BOOL; (* MCP PS4 전원 이상 *)
    MCP_M_PS_DC_LOW AT %MW353.0 : BOOL; (* MCP PS 전원 이상총괄 *)
    MCP_M_SAG1_1_이상 AT %MW352.1 : BOOL; (* MCP SAG장치 이상 *)
    MCP_M_SAG1_2_이상 AT %MW352.2 : BOOL; (* MC SAG장치2 이상 *)
    MCP_M_SAG_이상 AT %MW352.0 : BOOL; (* MCP SAG장치 이상총괄 *)
    MCP_M_SPD_이상 AT %MW354.0 : BOOL; (* MCP 동력반 SPD 이상 *)
    MCP_M_램프_테스트 AT %MW350.6 : BOOL; (* MCP SPB LAMP 테스트 *)
    MCP_M_부저_정지 AT %MW350.5 : BOOL; (* MCP 부저정지 *)
    MCP_M_비상정지 AT %MW350.7 : BOOL; (* MCP 비상정지 이상 *)
    MCP_M_비상정지_정상 AT %MW350.8 : BOOL;
    MCP_M_수동모드 AT %MW350.1 : BOOL; (* MCP ALL공정 수동모드 *)
    MCP_M_운전준비_ON AT %MW350.0 : BOOL; (* MCP ALL공정 운전준비 ON *)
    MCP_M_이상_리셋 AT %MW350.4 : BOOL; (* MCP PB 이상리셋 *)
    MCP_M_자동_운전중 AT %MW350.3 : BOOL; (* MCP ALL공정 자동운전중 *)
    MCP_M_자동모드 AT %MW350.2 : BOOL; (* MCP ALL공정 자동모드 *)
    MCP_M_총괄_이상 AT %MW302.0 : BOOL;
    MCP_M_통신_CP_TRIP AT %MW351.2 : BOOL; (* MCP   HMI전원  CP OFF 이상 *)
    MCP_M_통신_이상 AT %MW352.8 : BOOL; (* MCP 통신이상 *)
    R361_1_M_DATA_삭제_PLS AT %MW9000.0 : BOOL; (* R361 1 M DATA 삭제 PLS *)
    R361_1_M_DATA_삭제_SIGN AT %MW9000.1 : BOOL; (* R361 1 M DATA 삭제 SIGN *)
    R361_1_M_DATA_삭제_완료 AT %MW9000.2 : BOOL; (* R361 1 M DATA 삭제 완료 *)
    R361_1_M_NODE_4_01_통신_이상 AT %MW1524.8 : BOOL;
    R361_1_M_RACK3_동일차종 AT %MW1565.2 : BOOL;
    R361_1_M_RACK3_프로그램_OK AT %MW1563.2 : BOOL;
    R361_1_M_RACK4_동일차종 AT %MW1565.3 : BOOL;
    R361_1_M_RACK4_프로그램_OK AT %MW1563.3 : BOOL;
    R361_1_M_RACK5_동일차종 AT %MW1565.4 : BOOL;
    R361_1_M_RACK5_프로그램_OK AT %MW1563.4 : BOOL;
    R361_1_M_RACK6_동일차종 AT %MW1565.5 : BOOL;
    R361_1_M_RACK6_프로그램_OK AT %MW1563.5 : BOOL;
    R361_1_M_S365_DATA_전송_MEMO AT %MW9000.4 : BOOL; (* R361 1 M S365 DATA 전송 MEMO *)
    R361_1_M_S365_DATA_전송_PLS AT %MW9000.5 : BOOL; (* R361 1 M S365 DATA 전송 PLS *)
    R361_1_M_S365_DATA_전송_SIGN AT %MW9000.6 : BOOL; (* R361 1 M S365 DATA 전송 SIGN *)
    R361_1_M_S365_DATA_전송_완료 AT %MW9000.7 : BOOL; (* R361 1 M S365 DATA 전송 완료 *)
    R361_1_M_S366_DATA_전송_MEMO AT %MW9000.8 : BOOL; (* R361 1 M S366 DATA 전송 MEMO *)
    R361_1_M_S366_DATA_전송_PLS AT %MW9000.9 : BOOL; (* R361 1 M S366 DATA 전송 PLS *)
    R361_1_M_S366_DATA_전송_SIGN AT %MW9000.10 : BOOL; (* R361 1 M S366 DATA 전송 SIGN *)
    R361_1_M_S366_DATA_전송_완료 AT %MW9000.11 : BOOL; (* R361 1 M S366 DATA 전송 완료 *)
    R361_1_M_SEQ AT %MW10000 : WORD; (* R361 1 M SEQ *)
    R361_1_M_VIN_NO_1_2 AT %MW10011 : WORD; (* R361 1 M VIN NO 1 2 *)
    R361_1_M_VIN_NO_3_4 AT %MW10012 : WORD; (* R361 1 M VIN NO 3 4 *)
    R361_1_M_VIN_NO_5_6 AT %MW10013 : WORD; (* R361 1 M VIN NO 5 6 *)
    R361_1_M_VIN_NO_7_8 AT %MW10014 : WORD; (* R361 1 M VIN NO 7 8 *)
    R361_1_M_VIN_NO_9_10 AT %MW10015 : WORD; (* R361 1 M VIN NO 9 10 *)
    R361_1_M_공정_차종_유 : BOOL; (* S362_M_공정_차종_유 *)
    R361_1_M_기동_랙번호 AT %MW1534 : WORD;
    R361_1_M_부품비교차종 AT %MW1532 : WORD;
    R361_1_M_차종1_AX AT %MW10001.0 : BOOL; (* R361 1 M 차종1 AX *)
    R361_1_M_차종1_B AT %MW10001.1 : BOOL; (* R361 1 M 차종1 B *)
    R361_1_M_차종1_C AT %MW10001.2 : BOOL; (* R361 1 M 차종1 C *)
    R361_1_M_차종1_D AT %MW10001.3 : BOOL; (* R361 1 M 차종1 D *)
    R361_1_M_차종1_E AT %MW10001.4 : BOOL; (* R361 1 M 차종1 E *)
    R361_1_M_차종1_F AT %MW10001.5 : BOOL; (* R361 1 M 차종1 F *)
    R361_1_M_차종1_G AT %MW10001.6 : BOOL; (* R361 1 M 차종1 G *)
    R361_1_M_차종1_H AT %MW10001.7 : BOOL; (* R361 1 M 차종1 H *)
    R361_1_M_차종2_3DR AT %MW10001.8 : BOOL; (* R361 1 M 차종2 3DR *)
    R361_1_M_차종2_4DR AT %MW10001.9 : BOOL; (* R361 1 M 차종2 4DR *)
    R361_1_M_차종2_5DR AT %MW10001.10 : BOOL; (* R361 1 M 차종2 5DR *)
    R361_1_M_차종2_SP1 AT %MW10001.12 : BOOL; (* R361 1 M 차종2 SP1 *)
    R361_1_M_차종2_SP2 AT %MW10001.13 : BOOL; (* R361 1 M 차종2 SP2 *)
    R361_1_M_차종2_WGN AT %MW10001.11 : BOOL; (* R361 1 M 차종2 WGN *)
    R361_1_M_차종3_LHD AT %MW10001.14 : BOOL; (* R361 1 M 차종3 LHD *)
    R361_1_M_차종3_RHD AT %MW10001.15 : BOOL; (* R361 1 M 차종3 RHD *)
    R361_1_M_차종4_EEC AT %MW10002.3 : BOOL; (* R361 1 M 차종4 EEC *)
    R361_1_M_차종4_SP1 AT %MW10002.8 : BOOL; (* R361 1 M 차종4 SP1 *)
    R361_1_M_차종4_SP2 AT %MW10002.9 : BOOL; (* R361 1 M 차종4 SP2 *)
    R361_1_M_차종4_SP3 AT %MW10002.11 : BOOL; (* R361 1 M 차종4 SP3 *)
    R361_1_M_차종4_SP4 AT %MW10002.12 : BOOL; (* R361 1 M 차종4 SP4 *)
    R361_1_M_차종4_SP5 AT %MW10002.13 : BOOL; (* R361 1 M 차종4 SP5 *)
    R361_1_M_차종4_SP6 AT %MW10002.14 : BOOL; (* R361 1 M 차종4 SP6 *)
    R361_1_M_차종4_SP7 AT %MW10002.15 : BOOL; (* R361 1 M 차종4 SP7 *)
    R361_1_M_차종4_내수 AT %MW10002.0 : BOOL; (* R361 1 M 차종4 내수 *)
    R361_1_M_차종4_러시아 AT %MW10002.10 : BOOL; (* R361 1 M 차종4 러시아 *)
    R361_1_M_차종4_북미 AT %MW10002.2 : BOOL; (* R361 1 M 차종4 북미 *)
    R361_1_M_차종4_브라질 AT %MW10002.7 : BOOL; (* R361 1 M 차종4 브라질 *)
    R361_1_M_차종4_수출 AT %MW10002.1 : BOOL; (* R361 1 M 차종4 수출 *)
    R361_1_M_차종4_중국 AT %MW10002.6 : BOOL; (* R361 1 M 차종4 중국 *)
    R361_1_M_차종4_중동 AT %MW10002.5 : BOOL; (* R361 1 M 차종4 중동 *)
    R361_1_M_차종4_호주 AT %MW10002.4 : BOOL; (* R361 1 M 차종4 호주 *)
    R361_1_M_차종5_AT AT %MW10003.1 : BOOL; (* R361 1 M 차종5 AT *)
    R361_1_M_차종5_MT AT %MW10003.0 : BOOL; (* R361 1 M 차종5 MT *)
    R361_1_M_차종5_SP1 AT %MW10003.2 : BOOL; (* R361 1 M 차종5 SP1 *)
    R361_1_M_차종6_DSROOF AT %MW10003.6 : BOOL; (* R361 1 M 차종6 DSROOF *)
    R361_1_M_차종6_SP1 AT %MW10003.7 : BOOL; (* R361 1 M 차종6 SP1 *)
    R361_1_M_차종6_썬루프 AT %MW10003.4 : BOOL; (* R361 1 M 차종6 썬루프 *)
    R361_1_M_차종6_일반루프 AT %MW10003.3 : BOOL; (* R361 1 M 차종6 일반루프 *)
    R361_1_M_차종6_파노라마루프 AT %MW10003.5 : BOOL; (* R361 1 M 차종6 파노라마루프 *)
    R361_1_M_차종7_DSL AT %MW10003.9 : BOOL; (* R361 1 M 차종7 DSL *)
    R361_1_M_차종7_GSL AT %MW10003.8 : BOOL; (* R361 1 M 차종7 GSL *)
    R361_1_M_차종7_SP1 AT %MW10003.10 : BOOL; (* R361 1 M 차종7 SP1 *)
    R361_1_M_차종7_SP2 AT %MW10003.11 : BOOL; (* R361 1 M 차종7 SP2 *)
    R361_1_M_차종7_SP3 AT %MW10003.12 : BOOL; (* R361 1 M 차종7 SP3 *)
    R361_1_M_차종7_SP4 AT %MW10003.13 : BOOL; (* R361 1 M 차종7 SP4 *)
    R361_1_M_차종7_SP5 AT %MW10003.14 : BOOL; (* R361 1 M 차종7 SP5 *)
    R361_1_M_차종7_SP6 AT %MW10003.15 : BOOL; (* R361 1 M 차종7 SP6 *)
    R361_1_M_차종8_2WD AT %MW10004.0 : BOOL; (* R361 1 M 차종8 2WD *)
    R361_1_M_차종8_4WD AT %MW10004.1 : BOOL; (* R361 1 M 차종8 4WD *)
    R361_1_M_차종8_SP1 AT %MW10004.2 : BOOL; (* R361 1 M 차종8 SP1 *)
    R361_1_M_차종9_MPI AT %MW10004.3 : BOOL; (* R361 1 M 차종9 MPI *)
    R361_1_M_차종9_SP1 AT %MW10004.5 : BOOL; (* R361 1 M 차종9 SP1 *)
    R361_1_M_차종9_SP10 AT %MW10004.14 : BOOL; (* R361 1 M 차종9 SP10 *)
    R361_1_M_차종9_SP11 AT %MW10004.15 : BOOL; (* R361 1 M 차종9 SP11 *)
    R361_1_M_차종9_SP2 AT %MW10004.6 : BOOL; (* R361 1 M 차종9 SP2 *)
    R361_1_M_차종9_SP3 AT %MW10004.7 : BOOL; (* R361 1 M 차종9 SP3 *)
    R361_1_M_차종9_SP4 AT %MW10004.8 : BOOL; (* R361 1 M 차종9 SP4 *)
    R361_1_M_차종9_SP5 AT %MW10004.9 : BOOL; (* R361 1 M 차종9 SP5 *)
    R361_1_M_차종9_SP6 AT %MW10004.10 : BOOL; (* R361 1 M 차종9 SP6 *)
    R361_1_M_차종9_SP7 AT %MW10004.11 : BOOL; (* R361 1 M 차종9 SP7 *)
    R361_1_M_차종9_SP8 AT %MW10004.12 : BOOL; (* R361 1 M 차종9 SP8 *)
    R361_1_M_차종9_SP9 AT %MW10004.13 : BOOL; (* R361 1 M 차종9 SP9 *)
    R361_1_M_차종9_T_GDI AT %MW10004.4 : BOOL; (* R361 1 M 차종9 T GDI *)
    R361_1_M_차종_AS AT %MW10010.9 : BOOL; (* R361 1 M 차종 AS *)
    R361_1_M_차종_OPT1_R_RACK_무 AT %MW10005.3 : BOOL; (* R361 1 M 차종 OPT1 R RACK 무 *)
    R361_1_M_차종_OPT1_R_RACK_유 AT %MW10005.2 : BOOL; (* R361 1 M 차종 OPT1 R RACK 유 *)
    R361_1_M_차종_OPT1_SP1 AT %MW10005.10 : BOOL; (* R361 1 M 차종 OPT1 SP1 *)
    R361_1_M_차종_OPT1_SP2 AT %MW10005.11 : BOOL; (* R361 1 M 차종 OPT1 SP2 *)
    R361_1_M_차종_OPT1_SP3 AT %MW10005.12 : BOOL; (* R361 1 M 차종 OPT1 SP3 *)
    R361_1_M_차종_OPT1_SP4 AT %MW10005.13 : BOOL; (* R361 1 M 차종 OPT1 SP4 *)
    R361_1_M_차종_OPT1_SP5 AT %MW10005.14 : BOOL; (* R361 1 M 차종 OPT1 SP5 *)
    R361_1_M_차종_OPT1_SP6 AT %MW10005.15 : BOOL; (* R361 1 M 차종 OPT1 SP6 *)
    R361_1_M_차종_OPT1_S_REP_EATER_무 AT %MW10005.7 : BOOL; (* R361 1 M 차종 OPT1 S REP EATER 무 *)
    R361_1_M_차종_OPT1_S_REP_EATER_유 AT %MW10005.6 : BOOL; (* R361 1 M 차종 OPT1 S REP EATER 유 *)
    R361_1_M_차종_OPT1_VAN_무 AT %MW10005.9 : BOOL; (* R361 1 M 차종 OPT1 VAN 무 *)
    R361_1_M_차종_OPT1_VAN_유 AT %MW10005.8 : BOOL; (* R361 1 M 차종 OPT1 VAN 유 *)
    R361_1_M_차종_OPT1_슬라이딩_무 AT %MW10005.1 : BOOL; (* R361 1 M 차종 OPT1 슬라이딩 무 *)
    R361_1_M_차종_OPT1_슬라이딩_유 AT %MW10005.0 : BOOL; (* R361 1 M 차종 OPT1 슬라이딩 유 *)
    R361_1_M_차종_OPT1_폴딩_무 AT %MW10005.5 : BOOL; (* R361 1 M 차종 OPT1 폴딩 무 *)
    R361_1_M_차종_OPT1_폴딩_유 AT %MW10005.4 : BOOL; (* R361 1 M 차종 OPT1 폴딩 유 *)
    R361_1_M_차종_OPT2_SP_WORD1 AT %MW10006 : WORD; (* R361 1 M 차종 OPT2 SP WORD1 *)
    R361_1_M_차종_OPT3_SP_WORD2 AT %MW10007 : WORD; (* R361 1 M 차종 OPT3 SP WORD2 *)
    R361_1_M_차종_OPT4_SP_WORD3 AT %MW10008 : WORD; (* R361 1 M 차종 OPT4 SP WORD3 *)
    R361_1_M_차종_OPT5_SP_WORD4 AT %MW10009 : WORD; (* R361 1 M 차종 OPT5 SP WORD4 *)
    R361_1_M_차종_SP1 AT %MW10010.0 : BOOL; (* R361 1 M 차종 SP1 *)
    R361_1_M_차종_SP2 AT %MW10010.1 : BOOL; (* R361 1 M 차종 SP2 *)
    R361_1_M_차종_SP3 AT %MW10010.2 : BOOL; (* R361 1 M 차종 SP3 *)
    R361_1_M_차종_SP4 AT %MW10010.3 : BOOL; (* R361 1 M 차종 SP4 *)
    R361_1_M_차종_SP5 AT %MW10010.4 : BOOL; (* R361 1 M 차종 SP5 *)
    R361_1_M_차종_SP6 AT %MW10010.5 : BOOL; (* R361 1 M 차종 SP6 *)
    R361_1_M_차종_SP7 AT %MW10010.6 : BOOL; (* R361 1 M 차종 SP7 *)
    R361_1_M_차종_SP8 AT %MW10010.7 : BOOL; (* R361 1 M 차종 SP8 *)
    R361_1_M_차종_SP9 AT %MW10010.15 : BOOL; (* R361 1 M 차종 SP9 *)
    R361_1_M_차종_공대차 AT %MW10010.12 : BOOL; (* R361 1 M 차종 공대차 *)
    R361_1_M_차종_공차 AT %MW10010.10 : BOOL; (* R361 1 M 차종 공차 *)
    R361_1_M_차종_무 AT %MW1502.1 : BOOL;
    R361_1_M_차종_불량대차 AT %MW10010.13 : BOOL; (* R361 1 M 차종 불량대차 *)
    R361_1_M_차종_불량차 AT %MW10010.11 : BOOL; (* R361 1 M 차종 불량차 *)
    R361_1_M_차종_비축 AT %MW10010.8 : BOOL; (* R361 1 M 차종 비축 *)
    R361_1_M_차종_유 AT %MW1502.0 : BOOL;
    R361_1_M_차종_취출대차 AT %MW10010.14 : BOOL; (* R361 1 M 차종 취출대차 *)
    R361_2_M_DATA_삭제_PLS AT %MW9001.0 : BOOL; (* R361 2 M DATA 삭제 PLS *)
    R361_2_M_DATA_삭제_SIGN AT %MW9001.1 : BOOL; (* R361 2 M DATA 삭제 SIGN *)
    R361_2_M_DATA_삭제_완료 AT %MW9001.2 : BOOL; (* R361 2 M DATA 삭제 완료 *)
    R361_2_M_NODE_4_02_통신_이상 AT %MW1524.9 : BOOL;
    R361_2_M_R361_1_DATA_전송_MEMO AT %MW9001.8 : BOOL; (* R361 2 M R361 1 DATA 전송 MEMO *)
    R361_2_M_R361_1_DATA_전송_PLS AT %MW9001.9 : BOOL; (* R361 2 M R361 1 DATA 전송 PLS *)
    R361_2_M_R361_1_DATA_전송_SIGN AT %MW9001.10 : BOOL; (* R361 2 M R361 1 DATA 전송 SIGN *)
    R361_2_M_R361_1_DATA_전송_완료 AT %MW9001.11 : BOOL; (* R361 2 M R361 1 DATA 전송 완료 *)
    R361_2_M_RACK1_동일차종 AT %MW1565.0 : BOOL;
    R361_2_M_RACK1_프로그램_OK AT %MW1563.0 : BOOL;
    R361_2_M_RACK2_동일차종 AT %MW1565.1 : BOOL;
    R361_2_M_RACK2_프로그램_OK AT %MW1563.1 : BOOL;
    R361_2_M_S364_DATA_전송_MEMO AT %MW9001.4 : BOOL; (* R361 2 M S364 DATA 전송 MEMO *)
    R361_2_M_S364_DATA_전송_PLS AT %MW9001.5 : BOOL; (* R361 2 M S364 DATA 전송 PLS *)
    R361_2_M_S364_DATA_전송_SIG AT %MW9001.6 : BOOL; (* R361 2 M S364 DATA 전송 SIG *)
    R361_2_M_S364_DATA_전송_완료 AT %MW9001.7 : BOOL; (* R361 2 M S364 DATA 전송 완료 *)
    R361_2_M_SEQ AT %MW10020 : WORD; (* R361 2 M SEQ *)
    R361_2_M_VIN_NO_1_2 AT %MW10031 : WORD; (* R361 2 M VIN NO 1 2 *)
    R361_2_M_VIN_NO_3_4 AT %MW10032 : WORD; (* R361 2 M VIN NO 3 4 *)
    R361_2_M_VIN_NO_5_6 AT %MW10033 : WORD; (* R361 2 M VIN NO 5 6 *)
    R361_2_M_VIN_NO_7_8 AT %MW10034 : WORD; (* R361 2 M VIN NO 7 8 *)
    R361_2_M_VIN_NO_9_10 AT %MW10035 : WORD; (* R361 2 M VIN NO 9 10 *)
    R361_2_M_기동_랙번호 AT %MW1535 : WORD;
    R361_2_M_부품비교차종 AT %MW1533 : WORD;
    R361_2_M_차종1_AX AT %MW10021.0 : BOOL; (* R361 2 M 차종1 AX *)
    R361_2_M_차종1_B AT %MW10021.1 : BOOL; (* R361 2 M 차종1 B *)
    R361_2_M_차종1_C AT %MW10021.2 : BOOL; (* R361 2 M 차종1 C *)
    R361_2_M_차종1_D AT %MW10021.3 : BOOL; (* R361 2 M 차종1 D *)
    R361_2_M_차종1_E AT %MW10021.4 : BOOL; (* R361 2 M 차종1 E *)
    R361_2_M_차종1_F AT %MW10021.5 : BOOL; (* R361 2 M 차종1 F *)
    R361_2_M_차종1_G AT %MW10021.6 : BOOL; (* R361 2 M 차종1 G *)
    R361_2_M_차종1_H AT %MW10021.7 : BOOL; (* R361 2 M 차종1 H *)
    R361_2_M_차종2_3DR AT %MW10021.8 : BOOL; (* R361 2 M 차종2 3DR *)
    R361_2_M_차종2_4DR AT %MW10021.9 : BOOL; (* R361 2 M 차종2 4DR *)
    R361_2_M_차종2_5DR AT %MW10021.10 : BOOL; (* R361 2 M 차종2 5DR *)
    R361_2_M_차종2_SP1 AT %MW10021.12 : BOOL; (* R361 2 M 차종2 SP1 *)
    R361_2_M_차종2_SP2 AT %MW10021.13 : BOOL; (* R361 2 M 차종2 SP2 *)
    R361_2_M_차종2_WGN AT %MW10021.11 : BOOL; (* R361 2 M 차종2 WGN *)
    R361_2_M_차종3_LHD AT %MW10021.14 : BOOL; (* R361 2 M 차종3 LHD *)
    R361_2_M_차종3_RHD AT %MW10021.15 : BOOL; (* R361 2 M 차종3 RHD *)
    R361_2_M_차종4_EEC AT %MW10022.3 : BOOL; (* R361 2 M 차종4 EEC *)
    R361_2_M_차종4_SP1 AT %MW10022.8 : BOOL; (* R361 2 M 차종4 SP1 *)
    R361_2_M_차종4_SP2 AT %MW10022.9 : BOOL; (* R361 2 M 차종4 SP2 *)
    R361_2_M_차종4_SP3 AT %MW10022.11 : BOOL; (* R361 2 M 차종4 SP3 *)
    R361_2_M_차종4_SP4 AT %MW10022.12 : BOOL; (* R361 2 M 차종4 SP4 *)
    R361_2_M_차종4_SP5 AT %MW10022.13 : BOOL; (* R361 2 M 차종4 SP5 *)
    R361_2_M_차종4_SP6 AT %MW10022.14 : BOOL; (* R361 2 M 차종4 SP6 *)
    R361_2_M_차종4_SP7 AT %MW10022.15 : BOOL; (* R361 2 M 차종4 SP7 *)
    R361_2_M_차종4_내수 AT %MW10022.0 : BOOL; (* R361 2 M 차종4 내수 *)
    R361_2_M_차종4_러시아 AT %MW10022.10 : BOOL; (* R361 2 M 차종4 러시아 *)
    R361_2_M_차종4_북미 AT %MW10022.2 : BOOL; (* R361 2 M 차종4 북미 *)
    R361_2_M_차종4_브라질 AT %MW10022.7 : BOOL; (* R361 2 M 차종4 브라질 *)
    R361_2_M_차종4_수출 AT %MW10022.1 : BOOL; (* R361 2 M 차종4 수출 *)
    R361_2_M_차종4_중국 AT %MW10022.6 : BOOL; (* R361 2 M 차종4 중국 *)
    R361_2_M_차종4_중동 AT %MW10022.5 : BOOL; (* R361 2 M 차종4 중동 *)
    R361_2_M_차종4_호주 AT %MW10022.4 : BOOL; (* R361 2 M 차종4 호주 *)
    R361_2_M_차종5_AT AT %MW10023.1 : BOOL; (* R361 2 M 차종5 AT *)
    R361_2_M_차종5_MT AT %MW10023.0 : BOOL; (* R361 2 M 차종5 MT *)
    R361_2_M_차종5_SP1 AT %MW10023.2 : BOOL; (* R361 2 M 차종5 SP1 *)
    R361_2_M_차종6_DSROOF AT %MW10023.6 : BOOL; (* R361 2 M 차종6 DSROOF *)
    R361_2_M_차종6_SP1 AT %MW10023.7 : BOOL; (* R361 2 M 차종6 SP1 *)
    R361_2_M_차종6_썬루프 AT %MW10023.4 : BOOL; (* R361 2 M 차종6 썬루프 *)
    R361_2_M_차종6_일반루프 AT %MW10023.3 : BOOL; (* R361 2 M 차종6 일반루프 *)
    R361_2_M_차종6_파노라마루프 AT %MW10023.5 : BOOL; (* R361 2 M 차종6 파노라마루프 *)
    R361_2_M_차종7_DSL AT %MW10023.9 : BOOL; (* R361 2 M 차종7 DSL *)
    R361_2_M_차종7_GSL AT %MW10023.8 : BOOL; (* R361 2 M 차종7 GSL *)
    R361_2_M_차종7_SP1 AT %MW10023.10 : BOOL; (* R361 2 M 차종7 SP1 *)
    R361_2_M_차종7_SP2 AT %MW10023.11 : BOOL; (* R361 2 M 차종7 SP2 *)
    R361_2_M_차종7_SP3 AT %MW10023.12 : BOOL; (* R361 2 M 차종7 SP3 *)
    R361_2_M_차종7_SP4 AT %MW10023.13 : BOOL; (* R361 2 M 차종7 SP4 *)
    R361_2_M_차종7_SP5 AT %MW10023.14 : BOOL; (* R361 2 M 차종7 SP5 *)
    R361_2_M_차종7_SP6 AT %MW10023.15 : BOOL; (* R361 2 M 차종7 SP6 *)
    R361_2_M_차종8_2WD AT %MW10024.0 : BOOL; (* R361 2 M 차종8 2WD *)
    R361_2_M_차종8_4WD AT %MW10024.1 : BOOL; (* R361 2 M 차종8 4WD *)
    R361_2_M_차종8_SP1 AT %MW10024.2 : BOOL; (* R361 2 M 차종8 SP1 *)
    R361_2_M_차종9_MPI AT %MW10024.3 : BOOL; (* R361 2 M 차종9 MPI *)
    R361_2_M_차종9_SP1 AT %MW10024.5 : BOOL; (* R361 2 M 차종9 SP1 *)
    R361_2_M_차종9_SP10 AT %MW10024.14 : BOOL; (* R361 2 M 차종9 SP10 *)
    R361_2_M_차종9_SP11 AT %MW10024.15 : BOOL; (* R361 2 M 차종9 SP11 *)
    R361_2_M_차종9_SP2 AT %MW10024.6 : BOOL; (* R361 2 M 차종9 SP2 *)
    R361_2_M_차종9_SP3 AT %MW10024.7 : BOOL; (* R361 2 M 차종9 SP3 *)
    R361_2_M_차종9_SP4 AT %MW10024.8 : BOOL; (* R361 2 M 차종9 SP4 *)
    R361_2_M_차종9_SP5 AT %MW10024.9 : BOOL; (* R361 2 M 차종9 SP5 *)
    R361_2_M_차종9_SP6 AT %MW10024.10 : BOOL; (* R361 2 M 차종9 SP6 *)
    R361_2_M_차종9_SP7 AT %MW10024.11 : BOOL; (* R361 2 M 차종9 SP7 *)
    R361_2_M_차종9_SP8 AT %MW10024.12 : BOOL; (* R361 2 M 차종9 SP8 *)
    R361_2_M_차종9_SP9 AT %MW10024.13 : BOOL; (* R361 2 M 차종9 SP9 *)
    R361_2_M_차종9_T_GDI AT %MW10024.4 : BOOL; (* R361 2 M 차종9 T GDI *)
    R361_2_M_차종_AS AT %MW10030.9 : BOOL; (* R361 2 M 차종 AS *)
    R361_2_M_차종_OPT1_R_RACK_무 AT %MW10025.3 : BOOL; (* R361 2 M 차종 OPT1 R RACK 무 *)
    R361_2_M_차종_OPT1_R_RACK_유 AT %MW10025.2 : BOOL; (* R361 2 M 차종 OPT1 R RACK 유 *)
    R361_2_M_차종_OPT1_SP1 AT %MW10025.10 : BOOL; (* R361 2 M 차종 OPT1 SP1 *)
    R361_2_M_차종_OPT1_SP2 AT %MW10025.11 : BOOL; (* R361 2 M 차종 OPT1 SP2 *)
    R361_2_M_차종_OPT1_SP3 AT %MW10025.12 : BOOL; (* R361 2 M 차종 OPT1 SP3 *)
    R361_2_M_차종_OPT1_SP4 AT %MW10025.13 : BOOL; (* R361 2 M 차종 OPT1 SP4 *)
    R361_2_M_차종_OPT1_SP5 AT %MW10025.14 : BOOL; (* R361 2 M 차종 OPT1 SP5 *)
    R361_2_M_차종_OPT1_SP6 AT %MW10025.15 : BOOL; (* R361 2 M 차종 OPT1 SP6 *)
    R361_2_M_차종_OPT1_S_REP_EATER_무 AT %MW10025.7 : BOOL; (* R361 2 M 차종 OPT1 S REP EATER 무 *)
    R361_2_M_차종_OPT1_S_REP_EATER_유 AT %MW10025.6 : BOOL; (* R361 2 M 차종 OPT1 S REP EATER 유 *)
    R361_2_M_차종_OPT1_VAN_무 AT %MW10025.9 : BOOL; (* R361 2 M 차종 OPT1 VAN 무 *)
    R361_2_M_차종_OPT1_VAN_유 AT %MW10025.8 : BOOL; (* R361 2 M 차종 OPT1 VAN 유 *)
    R361_2_M_차종_OPT1_슬라이딩_무 AT %MW10025.1 : BOOL; (* R361 2 M 차종 OPT1 슬라이딩 무 *)
    R361_2_M_차종_OPT1_슬라이딩_유 AT %MW10025.0 : BOOL; (* R361 2 M 차종 OPT1 슬라이딩 유 *)
    R361_2_M_차종_OPT1_폴딩_무 AT %MW10025.5 : BOOL; (* R361 2 M 차종 OPT1 폴딩 무 *)
    R361_2_M_차종_OPT1_폴딩_유 AT %MW10025.4 : BOOL; (* R361 2 M 차종 OPT1 폴딩 유 *)
    R361_2_M_차종_OPT2_SP_WORD1 AT %MW10026 : WORD; (* R361 2 M 차종 OPT2 SP WORD1 *)
    R361_2_M_차종_OPT3_SP_WORD2 AT %MW10027 : WORD; (* R361 2 M 차종 OPT3 SP WORD2 *)
    R361_2_M_차종_OPT4_SP_WORD3 AT %MW10028 : WORD; (* R361 2 M 차종 OPT4 SP WORD3 *)
    R361_2_M_차종_OPT5_SP_WORD4 AT %MW10029 : WORD; (* R361 2 M 차종 OPT5 SP WORD4 *)
    R361_2_M_차종_SP1 AT %MW10030.0 : BOOL; (* R361 2 M 차종 SP1 *)
    R361_2_M_차종_SP2 AT %MW10030.1 : BOOL; (* R361 2 M 차종 SP2 *)
    R361_2_M_차종_SP3 AT %MW10030.2 : BOOL; (* R361 2 M 차종 SP3 *)
    R361_2_M_차종_SP4 AT %MW10030.3 : BOOL; (* R361 2 M 차종 SP4 *)
    R361_2_M_차종_SP5 AT %MW10030.4 : BOOL; (* R361 2 M 차종 SP5 *)
    R361_2_M_차종_SP6 AT %MW10030.5 : BOOL; (* R361 2 M 차종 SP6 *)
    R361_2_M_차종_SP7 AT %MW10030.6 : BOOL; (* R361 2 M 차종 SP7 *)
    R361_2_M_차종_SP8 AT %MW10030.7 : BOOL; (* R361 2 M 차종 SP8 *)
    R361_2_M_차종_SP9 AT %MW10030.15 : BOOL; (* R361 2 M 차종 SP9 *)
    R361_2_M_차종_공대차 AT %MW10030.12 : BOOL; (* R361 2 M 차종 공대차 *)
    R361_2_M_차종_공차 AT %MW10030.10 : BOOL; (* R361 2 M 차종 공차 *)
    R361_2_M_차종_무 AT %MW1502.3 : BOOL;
    R361_2_M_차종_불량대차 AT %MW10030.13 : BOOL; (* R361 2 M 차종 불량대차 *)
    R361_2_M_차종_불량차 AT %MW10030.11 : BOOL; (* R361 2 M 차종 불량차 *)
    R361_2_M_차종_비축 AT %MW10030.8 : BOOL; (* R361 2 M 차종 비축 *)
    R361_2_M_차종_유 AT %MW1502.2 : BOOL;
    R361_2_M_차종_취출대차 AT %MW10030.14 : BOOL; (* R361 2 M 차종 취출대차 *)
    R363_1_M_NODE_4_03_통신_이상 AT %MW1024.8 : BOOL;
    R363_2_M_DATA_삭제_PLS AT %MW9003.0 : BOOL; (* R363_2 M DATA 삭제 PLS *)
    R363_2_M_DATA_삭제_SIGN AT %MW9003.1 : BOOL; (* R363_2 M DATA 삭제 SIGN *)
    R363_2_M_DATA_삭제_완료 AT %MW9003.2 : BOOL; (* R363_2 M DATA 삭제 완료 *)
    R363_2_M_NODE_4_04_통신_이상 AT %MW1024.9 : BOOL;
    R363_2_M_S366_DATA_전송_MEMO AT %MW9003.8 : BOOL; (* R363_2 M S366 DATA 전송 MEMO *)
    R363_2_M_S366_DATA_전송_PLS AT %MW9003.9 : BOOL; (* R363_2 M S366 DATA 전송 PLS *)
    R363_2_M_S366_DATA_전송_SIGN AT %MW9003.10 : BOOL; (* R363_2 M S366 DATA 전송 SIGN *)
    R363_2_M_S366_DATA_전송_완료 AT %MW9003.11 : BOOL; (* R363_2 M S366 DATA 전송 완료 *)
    R363_2_M_SEQ AT %MW10040 : WORD; (* R363 2 M SEQ *)
    R363_2_M_VIN_NO_1_2 AT %MW10051 : WORD; (* R363 2 M VIN NO 1 2 *)
    R363_2_M_VIN_NO_3_4 AT %MW10052 : WORD; (* R363 2 M VIN NO 3 4 *)
    R363_2_M_VIN_NO_5_6 AT %MW10053 : WORD; (* R363 2 M VIN NO 5 6 *)
    R363_2_M_VIN_NO_7_8 AT %MW10054 : WORD; (* R363 2 M VIN NO 7 8 *)
    R363_2_M_VIN_NO_9_10 AT %MW10055 : WORD; (* R363 2 M VIN NO 9 10 *)
    R363_2_M_차종1_AX AT %MW10041.0 : BOOL; (* R363 2 M 차종1 AX *)
    R363_2_M_차종1_B AT %MW10041.1 : BOOL; (* R363 2 M 차종1 B *)
    R363_2_M_차종1_C AT %MW10041.2 : BOOL; (* R363 2 M 차종1 C *)
    R363_2_M_차종1_D AT %MW10041.3 : BOOL; (* R363 2 M 차종1 D *)
    R363_2_M_차종1_E AT %MW10041.4 : BOOL; (* R363 2 M 차종1 E *)
    R363_2_M_차종1_F AT %MW10041.5 : BOOL; (* R363 2 M 차종1 F *)
    R363_2_M_차종1_G AT %MW10041.6 : BOOL; (* R363 2 M 차종1 G *)
    R363_2_M_차종1_H AT %MW10041.7 : BOOL; (* R363 2 M 차종1 H *)
    R363_2_M_차종2_3DR AT %MW10041.8 : BOOL; (* R363 2 M 차종2 3DR *)
    R363_2_M_차종2_4DR AT %MW10041.9 : BOOL; (* R363 2 M 차종2 4DR *)
    R363_2_M_차종2_5DR AT %MW10041.10 : BOOL; (* R363 2 M 차종2 5DR *)
    R363_2_M_차종2_SP1 AT %MW10041.12 : BOOL; (* R363 2 M 차종2 SP1 *)
    R363_2_M_차종2_SP2 AT %MW10041.13 : BOOL; (* R363 2 M 차종2 SP2 *)
    R363_2_M_차종2_WGN AT %MW10041.11 : BOOL; (* R363 2 M 차종2 WGN *)
    R363_2_M_차종3_LHD AT %MW10041.14 : BOOL; (* R363 2 M 차종3 LHD *)
    R363_2_M_차종3_RHD AT %MW10041.15 : BOOL; (* R363 2 M 차종3 RHD *)
    R363_2_M_차종4_EEC AT %MW10042.3 : BOOL; (* R363 2 M 차종4 EEC *)
    R363_2_M_차종4_SP1 AT %MW10042.8 : BOOL; (* R363 2 M 차종4 SP1 *)
    R363_2_M_차종4_SP2 AT %MW10042.9 : BOOL; (* R363 2 M 차종4 SP2 *)
    R363_2_M_차종4_SP3 AT %MW10042.11 : BOOL; (* R363 2 M 차종4 SP3 *)
    R363_2_M_차종4_SP4 AT %MW10042.12 : BOOL; (* R363 2 M 차종4 SP4 *)
    R363_2_M_차종4_SP5 AT %MW10042.13 : BOOL; (* R363 2 M 차종4 SP5 *)
    R363_2_M_차종4_SP6 AT %MW10042.14 : BOOL; (* R363 2 M 차종4 SP6 *)
    R363_2_M_차종4_SP7 AT %MW10042.15 : BOOL; (* R363 2 M 차종4 SP7 *)
    R363_2_M_차종4_내수 AT %MW10042.0 : BOOL; (* R363 2 M 차종4 내수 *)
    R363_2_M_차종4_러시아 AT %MW10042.10 : BOOL; (* R363 2 M 차종4 러시아 *)
    R363_2_M_차종4_북미 AT %MW10042.2 : BOOL; (* R363 2 M 차종4 북미 *)
    R363_2_M_차종4_브라질 AT %MW10042.7 : BOOL; (* R363 2 M 차종4 브라질 *)
    R363_2_M_차종4_수출 AT %MW10042.1 : BOOL; (* R363 2 M 차종4 수출 *)
    R363_2_M_차종4_중국 AT %MW10042.6 : BOOL; (* R363 2 M 차종4 중국 *)
    R363_2_M_차종4_중동 AT %MW10042.5 : BOOL; (* R363 2 M 차종4 중동 *)
    R363_2_M_차종4_호주 AT %MW10042.4 : BOOL; (* R363 2 M 차종4 호주 *)
    R363_2_M_차종5_AT AT %MW10043.1 : BOOL; (* R363 2 M 차종5 AT *)
    R363_2_M_차종5_MT AT %MW10043.0 : BOOL; (* R363 2 M 차종5 MT *)
    R363_2_M_차종5_SP1 AT %MW10043.2 : BOOL; (* R363 2 M 차종5 SP1 *)
    R363_2_M_차종6_DSROOF AT %MW10043.6 : BOOL; (* R363 2 M 차종6 DSROOF *)
    R363_2_M_차종6_SP1 AT %MW10043.7 : BOOL; (* R363 2 M 차종6 SP1 *)
    R363_2_M_차종6_썬루프 AT %MW10043.4 : BOOL; (* R363 2 M 차종6 썬루프 *)
    R363_2_M_차종6_일반루프 AT %MW10043.3 : BOOL; (* R363 2 M 차종6 일반루프 *)
    R363_2_M_차종6_파노라마루프 AT %MW10043.5 : BOOL; (* R363 2 M 차종6 파노라마루프 *)
    R363_2_M_차종7_DSL AT %MW10043.9 : BOOL; (* R363 2 M 차종7 DSL *)
    R363_2_M_차종7_GSL AT %MW10043.8 : BOOL; (* R363 2 M 차종7 GSL *)
    R363_2_M_차종7_SP1 AT %MW10043.10 : BOOL; (* R363 2 M 차종7 SP1 *)
    R363_2_M_차종7_SP2 AT %MW10043.11 : BOOL; (* R363 2 M 차종7 SP2 *)
    R363_2_M_차종7_SP3 AT %MW10043.12 : BOOL; (* R363 2 M 차종7 SP3 *)
    R363_2_M_차종7_SP4 AT %MW10043.13 : BOOL; (* R363 2 M 차종7 SP4 *)
    R363_2_M_차종7_SP5 AT %MW10043.14 : BOOL; (* R363 2 M 차종7 SP5 *)
    R363_2_M_차종7_SP6 AT %MW10043.15 : BOOL; (* R363 2 M 차종7 SP6 *)
    R363_2_M_차종8_2WD AT %MW10044.0 : BOOL; (* R363 2 M 차종8 2WD *)
    R363_2_M_차종8_4WD AT %MW10044.1 : BOOL; (* R363 2 M 차종8 4WD *)
    R363_2_M_차종8_SP1 AT %MW10044.2 : BOOL; (* R363 2 M 차종8 SP1 *)
    R363_2_M_차종9_MPI AT %MW10044.3 : BOOL; (* R363 2 M 차종9 MPI *)
    R363_2_M_차종9_SP1 AT %MW10044.5 : BOOL; (* R363 2 M 차종9 SP1 *)
    R363_2_M_차종9_SP10 AT %MW10044.14 : BOOL; (* R363 2 M 차종9 SP10 *)
    R363_2_M_차종9_SP11 AT %MW10044.15 : BOOL; (* R363 2 M 차종9 SP11 *)
    R363_2_M_차종9_SP2 AT %MW10044.6 : BOOL; (* R363 2 M 차종9 SP2 *)
    R363_2_M_차종9_SP3 AT %MW10044.7 : BOOL; (* R363 2 M 차종9 SP3 *)
    R363_2_M_차종9_SP4 AT %MW10044.8 : BOOL; (* R363 2 M 차종9 SP4 *)
    R363_2_M_차종9_SP5 AT %MW10044.9 : BOOL; (* R363 2 M 차종9 SP5 *)
    R363_2_M_차종9_SP6 AT %MW10044.10 : BOOL; (* R363 2 M 차종9 SP6 *)
    R363_2_M_차종9_SP7 AT %MW10044.11 : BOOL; (* R363 2 M 차종9 SP7 *)
    R363_2_M_차종9_SP8 AT %MW10044.12 : BOOL; (* R363 2 M 차종9 SP8 *)
    R363_2_M_차종9_SP9 AT %MW10044.13 : BOOL; (* R363 2 M 차종9 SP9 *)
    R363_2_M_차종9_T_GDI AT %MW10044.4 : BOOL; (* R363 2 M 차종9 T GDI *)
    R363_2_M_차종_AS AT %MW10050.9 : BOOL; (* R363 2 M 차종 AS *)
    R363_2_M_차종_OPT1_R_RACK_무 AT %MW10045.3 : BOOL; (* R363 2 M 차종 OPT1 R RACK 무 *)
    R363_2_M_차종_OPT1_R_RACK_유 AT %MW10045.2 : BOOL; (* R363 2 M 차종 OPT1 R RACK 유 *)
    R363_2_M_차종_OPT1_SP1 AT %MW10045.10 : BOOL; (* R363 2 M 차종 OPT1 SP1 *)
    R363_2_M_차종_OPT1_SP2 AT %MW10045.11 : BOOL; (* R363 2 M 차종 OPT1 SP2 *)
    R363_2_M_차종_OPT1_SP3 AT %MW10045.12 : BOOL; (* R363 2 M 차종 OPT1 SP3 *)
    R363_2_M_차종_OPT1_SP4 AT %MW10045.13 : BOOL; (* R363 2 M 차종 OPT1 SP4 *)
    R363_2_M_차종_OPT1_SP5 AT %MW10045.14 : BOOL; (* R363 2 M 차종 OPT1 SP5 *)
    R363_2_M_차종_OPT1_SP6 AT %MW10045.15 : BOOL; (* R363 2 M 차종 OPT1 SP6 *)
    R363_2_M_차종_OPT1_S_REP_EATER_무 AT %MW10045.7 : BOOL; (* R363 2 M 차종 OPT1 S REP EATER 무 *)
    R363_2_M_차종_OPT1_S_REP_EATER_유 AT %MW10045.6 : BOOL; (* R363 2 M 차종 OPT1 S REP EATER 유 *)
    R363_2_M_차종_OPT1_VAN_무 AT %MW10045.9 : BOOL; (* R363 2 M 차종 OPT1 VAN 무 *)
    R363_2_M_차종_OPT1_VAN_유 AT %MW10045.8 : BOOL; (* R363 2 M 차종 OPT1 VAN 유 *)
    R363_2_M_차종_OPT1_슬라이딩_무 AT %MW10045.1 : BOOL; (* R363 2 M 차종 OPT1 슬라이딩 무 *)
    R363_2_M_차종_OPT1_슬라이딩_유 AT %MW10045.0 : BOOL; (* R363 2 M 차종 OPT1 슬라이딩 유 *)
    R363_2_M_차종_OPT1_폴딩_무 AT %MW10045.5 : BOOL; (* R363 2 M 차종 OPT1 폴딩 무 *)
    R363_2_M_차종_OPT1_폴딩_유 AT %MW10045.4 : BOOL; (* R363 2 M 차종 OPT1 폴딩 유 *)
    R363_2_M_차종_OPT2_SP_WORD1 AT %MW10046 : WORD; (* R363 2 M 차종 OPT2 SP WORD1 *)
    R363_2_M_차종_OPT3_SP_WORD2 AT %MW10047 : WORD; (* R363 2 M 차종 OPT3 SP WORD2 *)
    R363_2_M_차종_OPT4_SP_WORD3 AT %MW10048 : WORD; (* R363 2 M 차종 OPT4 SP WORD3 *)
    R363_2_M_차종_OPT5_SP_WORD4 AT %MW10049 : WORD; (* R363 2 M 차종 OPT5 SP WORD4 *)
    R363_2_M_차종_SP1 AT %MW10050.0 : BOOL; (* R363 2 M 차종 SP1 *)
    R363_2_M_차종_SP2 AT %MW10050.1 : BOOL; (* R363 2 M 차종 SP2 *)
    R363_2_M_차종_SP3 AT %MW10050.2 : BOOL; (* R363 2 M 차종 SP3 *)
    R363_2_M_차종_SP4 AT %MW10050.3 : BOOL; (* R363 2 M 차종 SP4 *)
    R363_2_M_차종_SP5 AT %MW10050.4 : BOOL; (* R363 2 M 차종 SP5 *)
    R363_2_M_차종_SP6 AT %MW10050.5 : BOOL; (* R363 2 M 차종 SP6 *)
    R363_2_M_차종_SP7 AT %MW10050.6 : BOOL; (* R363 2 M 차종 SP7 *)
    R363_2_M_차종_SP8 AT %MW10050.7 : BOOL; (* R363 2 M 차종 SP8 *)
    R363_2_M_차종_SP9 AT %MW10050.15 : BOOL; (* R363 2 M 차종 SP9 *)
    R363_2_M_차종_공대차 AT %MW10050.12 : BOOL; (* R363 2 M 차종 공대차 *)
    R363_2_M_차종_공차 AT %MW10050.10 : BOOL; (* R363 2 M 차종 공차 *)
    R363_2_M_차종_무 AT %MW1002.3 : BOOL;
    R363_2_M_차종_불량대차 AT %MW10050.13 : BOOL; (* R363 2 M 차종 불량대차 *)
    R363_2_M_차종_불량차 AT %MW10050.11 : BOOL; (* R363 2 M 차종 불량차 *)
    R363_2_M_차종_비축 AT %MW10050.8 : BOOL; (* R363 2 M 차종 비축 *)
    R363_2_M_차종_유 AT %MW1002.2 : BOOL; (* S362_M_공정_차종_보조 *)
    R363_2_M_차종_취출대차 AT %MW10050.14 : BOOL; (* R363 2 M 차종 취출대차 *)
    R364_1_M_AX_차종_용접타점수 AT %MW8010 : WORD;
    R364_1_M_NODE_4_05_통신_이상 AT %MW2024.8 : BOOL;
    R364_1_M_용접_카운트_이상 AT %MW2029.0 : BOOL;
    R364_1_M_용접완료 AT %MW2006.1 : BOOL;
    R364_1_M_용접타점수_OK AT %MW2006.8 : BOOL;
    R366_1_M_AX_차종_용접타점수 AT %MW8060 : WORD;
    R366_1_M_NODE_4_06_통신_이상 AT %MW3024.8 : BOOL;
    R366_1_M_용접_카운트_이상 AT %MW3029.0 : BOOL;
    R366_1_M_용접완료 AT %MW3006.1 : BOOL;
    R366_1_M_용접타점수_OK AT %MW3006.8 : BOOL;
    R368_1_M_NODE_4_07_통신_이상 AT %MW4024.8 : BOOL;
    R369_1_M_DATA_삭제_PLS AT %MW9007.0 : BOOL; (* R369 1 M DATA 삭제 PLS *)
    R369_1_M_DATA_삭제_SIGN AT %MW9007.1 : BOOL; (* R369 1 M DATA 삭제 SIGN *)
    R369_1_M_DATA_삭제_완료 AT %MW9007.2 : BOOL; (* R369 1 M DATA 삭제 완료 *)
    R369_1_M_NODE_4_08_통신_이상 AT %MW4524.8 : BOOL;
    R369_1_M_S368_DATA_전송_MEMO AT %MW9007.4 : BOOL; (* R369 1 M S368 DATA 전송 MEMO *)
    R369_1_M_S368_DATA_전송_PLS AT %MW9007.5 : BOOL; (* R369 1 M S368 DATA 전송 PLS *)
    R369_1_M_S368_DATA_전송_SIGN AT %MW9007.6 : BOOL; (* R369 1 M S368 DATA 전송 SIGN *)
    R369_1_M_S368_DATA_전송_완료 AT %MW9007.7 : BOOL; (* R369 1 M S368 DATA 전송 완료 *)
    R369_1_M_S369_1_DATA_전송_MEMO AT %MW9007.8 : BOOL; (* R369 1 M S369 1 DATA 전송 MEMO *)
    R369_1_M_S369_1_DATA_전송_PLS AT %MW9007.9 : BOOL; (* R369 1 M S369 1 DATA 전송 PLS *)
    R369_1_M_S369_1_DATA_전송_SIGN AT %MW9007.10 : BOOL; (* R369 1 M S369 1 DATA 전송 SIGN *)
    R369_1_M_S369_1_DATA_전송_완료 AT %MW9007.11 : BOOL; (* R369 1 M S369 1 DATA 전송 완료 *)
    R369_1_M_SEQ AT %MW10060 : WORD; (* R369 1 M SEQ *)
    R369_1_M_VIN_NO_1_2 AT %MW10071 : WORD; (* R369 1 M VIN NO 1 2 *)
    R369_1_M_VIN_NO_3_4 AT %MW10072 : WORD; (* R369 1 M VIN NO 3 4 *)
    R369_1_M_VIN_NO_5_6 AT %MW10073 : WORD; (* R369 1 M VIN NO 5 6 *)
    R369_1_M_VIN_NO_7_8 AT %MW10074 : WORD; (* R369 1 M VIN NO 7 8 *)
    R369_1_M_VIN_NO_9_10 AT %MW10075 : WORD; (* R369 1 M VIN NO 9 10 *)
    R369_1_M_차종1_AX AT %MW10061.0 : BOOL; (* R369 1 M 차종1 AX *)
    R369_1_M_차종1_B AT %MW10061.1 : BOOL; (* R369 1 M 차종1 B *)
    R369_1_M_차종1_C AT %MW10061.2 : BOOL; (* R369 1 M 차종1 C *)
    R369_1_M_차종1_D AT %MW10061.3 : BOOL; (* R369 1 M 차종1 D *)
    R369_1_M_차종1_E AT %MW10061.4 : BOOL; (* R369 1 M 차종1 E *)
    R369_1_M_차종1_F AT %MW10061.5 : BOOL; (* R369 1 M 차종1 F *)
    R369_1_M_차종1_G AT %MW10061.6 : BOOL; (* R369 1 M 차종1 G *)
    R369_1_M_차종1_H AT %MW10061.7 : BOOL; (* R369 1 M 차종1 H *)
    R369_1_M_차종2_3DR AT %MW10061.8 : BOOL; (* R369 1 M 차종2 3DR *)
    R369_1_M_차종2_4DR AT %MW10061.9 : BOOL; (* R369 1 M 차종2 4DR *)
    R369_1_M_차종2_5DR AT %MW10061.10 : BOOL; (* R369 1 M 차종2 5DR *)
    R369_1_M_차종2_SP1 AT %MW10061.12 : BOOL; (* R369 1 M 차종2 SP1 *)
    R369_1_M_차종2_SP2 AT %MW10061.13 : BOOL; (* R369 1 M 차종2 SP2 *)
    R369_1_M_차종2_WGN AT %MW10061.11 : BOOL; (* R369 1 M 차종2 WGN *)
    R369_1_M_차종3_LHD AT %MW10061.14 : BOOL; (* R369 1 M 차종3 LHD *)
    R369_1_M_차종3_RHD AT %MW10061.15 : BOOL; (* R369 1 M 차종3 RHD *)
    R369_1_M_차종4_EEC AT %MW10062.3 : BOOL; (* R369 1 M 차종4 EEC *)
    R369_1_M_차종4_SP1 AT %MW10062.8 : BOOL; (* R369 1 M 차종4 SP1 *)
    R369_1_M_차종4_SP2 AT %MW10062.9 : BOOL; (* R369 1 M 차종4 SP2 *)
    R369_1_M_차종4_SP3 AT %MW10062.11 : BOOL; (* R369 1 M 차종4 SP3 *)
    R369_1_M_차종4_SP4 AT %MW10062.12 : BOOL; (* R369 1 M 차종4 SP4 *)
    R369_1_M_차종4_SP5 AT %MW10062.13 : BOOL; (* R369 1 M 차종4 SP5 *)
    R369_1_M_차종4_SP6 AT %MW10062.14 : BOOL; (* R369 1 M 차종4 SP6 *)
    R369_1_M_차종4_SP7 AT %MW10062.15 : BOOL; (* R369 1 M 차종4 SP7 *)
    R369_1_M_차종4_내수 AT %MW10062.0 : BOOL; (* R369 1 M 차종4 내수 *)
    R369_1_M_차종4_러시아 AT %MW10062.10 : BOOL; (* R369 1 M 차종4 러시아 *)
    R369_1_M_차종4_북미 AT %MW10062.2 : BOOL; (* R369 1 M 차종4 북미 *)
    R369_1_M_차종4_브라질 AT %MW10062.7 : BOOL; (* R369 1 M 차종4 브라질 *)
    R369_1_M_차종4_수출 AT %MW10062.1 : BOOL; (* R369 1 M 차종4 수출 *)
    R369_1_M_차종4_중국 AT %MW10062.6 : BOOL; (* R369 1 M 차종4 중국 *)
    R369_1_M_차종4_중동 AT %MW10062.5 : BOOL; (* R369 1 M 차종4 중동 *)
    R369_1_M_차종4_호주 AT %MW10062.4 : BOOL; (* R369 1 M 차종4 호주 *)
    R369_1_M_차종5_AT AT %MW10063.1 : BOOL; (* R369 1 M 차종5 AT *)
    R369_1_M_차종5_MT AT %MW10063.0 : BOOL; (* R369 1 M 차종5 MT *)
    R369_1_M_차종5_SP1 AT %MW10063.2 : BOOL; (* R369 1 M 차종5 SP1 *)
    R369_1_M_차종6_DSROOF AT %MW10063.6 : BOOL; (* R369 1 M 차종6 DSROOF *)
    R369_1_M_차종6_SP1 AT %MW10063.7 : BOOL; (* R369 1 M 차종6 SP1 *)
    R369_1_M_차종6_썬루프 AT %MW10063.4 : BOOL; (* R369 1 M 차종6 썬루프 *)
    R369_1_M_차종6_일반루프 AT %MW10063.3 : BOOL; (* R369 1 M 차종6 일반루프 *)
    R369_1_M_차종6_파노라마루프 AT %MW10063.5 : BOOL; (* R369 1 M 차종6 파노라마루프 *)
    R369_1_M_차종7_DSL AT %MW10063.9 : BOOL; (* R369 1 M 차종7 DSL *)
    R369_1_M_차종7_GSL AT %MW10063.8 : BOOL; (* R369 1 M 차종7 GSL *)
    R369_1_M_차종7_SP1 AT %MW10063.10 : BOOL; (* R369 1 M 차종7 SP1 *)
    R369_1_M_차종7_SP2 AT %MW10063.11 : BOOL; (* R369 1 M 차종7 SP2 *)
    R369_1_M_차종7_SP3 AT %MW10063.12 : BOOL; (* R369 1 M 차종7 SP3 *)
    R369_1_M_차종7_SP4 AT %MW10063.13 : BOOL; (* R369 1 M 차종7 SP4 *)
    R369_1_M_차종7_SP5 AT %MW10063.14 : BOOL; (* R369 1 M 차종7 SP5 *)
    R369_1_M_차종7_SP6 AT %MW10063.15 : BOOL; (* R369 1 M 차종7 SP6 *)
    R369_1_M_차종8_2WD AT %MW10064.0 : BOOL; (* R369 1 M 차종8 2WD *)
    R369_1_M_차종8_4WD AT %MW10064.1 : BOOL; (* R369 1 M 차종8 4WD *)
    R369_1_M_차종8_SP1 AT %MW10064.2 : BOOL; (* R369 1 M 차종8 SP1 *)
    R369_1_M_차종9_MPI AT %MW10064.3 : BOOL; (* R369 1 M 차종9 MPI *)
    R369_1_M_차종9_SP1 AT %MW10064.5 : BOOL; (* R369 1 M 차종9 SP1 *)
    R369_1_M_차종9_SP10 AT %MW10064.14 : BOOL; (* R369 1 M 차종9 SP10 *)
    R369_1_M_차종9_SP11 AT %MW10064.15 : BOOL; (* R369 1 M 차종9 SP11 *)
    R369_1_M_차종9_SP2 AT %MW10064.6 : BOOL; (* R369 1 M 차종9 SP2 *)
    R369_1_M_차종9_SP3 AT %MW10064.7 : BOOL; (* R369 1 M 차종9 SP3 *)
    R369_1_M_차종9_SP4 AT %MW10064.8 : BOOL; (* R369 1 M 차종9 SP4 *)
    R369_1_M_차종9_SP5 AT %MW10064.9 : BOOL; (* R369 1 M 차종9 SP5 *)
    R369_1_M_차종9_SP6 AT %MW10064.10 : BOOL; (* R369 1 M 차종9 SP6 *)
    R369_1_M_차종9_SP7 AT %MW10064.11 : BOOL; (* R369 1 M 차종9 SP7 *)
    R369_1_M_차종9_SP8 AT %MW10064.12 : BOOL; (* R369 1 M 차종9 SP8 *)
    R369_1_M_차종9_SP9 AT %MW10064.13 : BOOL; (* R369 1 M 차종9 SP9 *)
    R369_1_M_차종9_T_GDI AT %MW10064.4 : BOOL; (* R369 1 M 차종9 T GDI *)
    R369_1_M_차종_AS AT %MW10070.9 : BOOL; (* R369 1 M 차종 AS *)
    R369_1_M_차종_OPT1_R_RACK_무 AT %MW10065.3 : BOOL; (* R369 1 M 차종 OPT1 R RACK 무 *)
    R369_1_M_차종_OPT1_R_RACK_유 AT %MW10065.2 : BOOL; (* R369 1 M 차종 OPT1 R RACK 유 *)
    R369_1_M_차종_OPT1_SP1 AT %MW10065.10 : BOOL; (* R369 1 M 차종 OPT1 SP1 *)
    R369_1_M_차종_OPT1_SP2 AT %MW10065.11 : BOOL; (* R369 1 M 차종 OPT1 SP2 *)
    R369_1_M_차종_OPT1_SP3 AT %MW10065.12 : BOOL; (* R369 1 M 차종 OPT1 SP3 *)
    R369_1_M_차종_OPT1_SP4 AT %MW10065.13 : BOOL; (* R369 1 M 차종 OPT1 SP4 *)
    R369_1_M_차종_OPT1_SP5 AT %MW10065.14 : BOOL; (* R369 1 M 차종 OPT1 SP5 *)
    R369_1_M_차종_OPT1_SP6 AT %MW10065.15 : BOOL; (* R369 1 M 차종 OPT1 SP6 *)
    R369_1_M_차종_OPT1_S_REP_EATER_무 AT %MW10065.7 : BOOL; (* R369 1 M 차종 OPT1 S REP EATER 무 *)
    R369_1_M_차종_OPT1_S_REP_EATER_유 AT %MW10065.6 : BOOL; (* R369 1 M 차종 OPT1 S REP EATER 유 *)
    R369_1_M_차종_OPT1_VAN_무 AT %MW10065.9 : BOOL; (* R369 1 M 차종 OPT1 VAN 무 *)
    R369_1_M_차종_OPT1_VAN_유 AT %MW10065.8 : BOOL; (* R369 1 M 차종 OPT1 VAN 유 *)
    R369_1_M_차종_OPT1_슬라이딩_무 AT %MW10065.1 : BOOL; (* R369 1 M 차종 OPT1 슬라이딩 무 *)
    R369_1_M_차종_OPT1_슬라이딩_유 AT %MW10065.0 : BOOL; (* R369 1 M 차종 OPT1 슬라이딩 유 *)
    R369_1_M_차종_OPT1_폴딩_무 AT %MW10065.5 : BOOL; (* R369 1 M 차종 OPT1 폴딩 무 *)
    R369_1_M_차종_OPT1_폴딩_유 AT %MW10065.4 : BOOL; (* R369 1 M 차종 OPT1 폴딩 유 *)
    R369_1_M_차종_OPT2_SP_WORD1 AT %MW10066 : WORD; (* R369 1 M 차종 OPT2 SP WORD1 *)
    R369_1_M_차종_OPT3_SP_WORD2 AT %MW10067 : WORD; (* R369 1 M 차종 OPT3 SP WORD2 *)
    R369_1_M_차종_OPT4_SP_WORD3 AT %MW10068 : WORD; (* R369 1 M 차종 OPT4 SP WORD3 *)
    R369_1_M_차종_OPT5_SP_WORD4 AT %MW10069 : WORD; (* R369 1 M 차종 OPT5 SP WORD4 *)
    R369_1_M_차종_SP1 AT %MW10070.0 : BOOL; (* R369 1 M 차종 SP1 *)
    R369_1_M_차종_SP2 AT %MW10070.1 : BOOL; (* R369 1 M 차종 SP2 *)
    R369_1_M_차종_SP3 AT %MW10070.2 : BOOL; (* R369 1 M 차종 SP3 *)
    R369_1_M_차종_SP4 AT %MW10070.3 : BOOL; (* R369 1 M 차종 SP4 *)
    R369_1_M_차종_SP5 AT %MW10070.4 : BOOL; (* R369 1 M 차종 SP5 *)
    R369_1_M_차종_SP6 AT %MW10070.5 : BOOL; (* R369 1 M 차종 SP6 *)
    R369_1_M_차종_SP7 AT %MW10070.6 : BOOL; (* R369 1 M 차종 SP7 *)
    R369_1_M_차종_SP8 AT %MW10070.7 : BOOL; (* R369 1 M 차종 SP8 *)
    R369_1_M_차종_SP9 AT %MW10070.15 : BOOL; (* R369 1 M 차종 SP9 *)
    R369_1_M_차종_공대차 AT %MW10070.12 : BOOL; (* R369 1 M 차종 공대차 *)
    R369_1_M_차종_공차 AT %MW10070.10 : BOOL; (* R369 1 M 차종 공차 *)
    R369_1_M_차종_무 AT %MW4502.3 : BOOL;
    R369_1_M_차종_불량대차 AT %MW10070.13 : BOOL; (* R369 1 M 차종 불량대차 *)
    R369_1_M_차종_불량차 AT %MW10070.11 : BOOL; (* R369 1 M 차종 불량차 *)
    R369_1_M_차종_비축 AT %MW10070.8 : BOOL; (* R369 1 M 차종 비축 *)
    R369_1_M_차종_유 AT %MW4502.2 : BOOL;
    R369_1_M_차종_취출대차 AT %MW10070.14 : BOOL; (* R369 1 M 차종 취출대차 *)
    R369_2_M_DATA_삭제_PLS AT %MW9008.0 : BOOL; (* R369 2 M DATA 삭제 PLS *)
    R369_2_M_DATA_삭제_SIGN AT %MW9008.1 : BOOL; (* R369 2 M DATA 삭제 SIGN *)
    R369_2_M_DATA_삭제_완료 AT %MW9008.2 : BOOL; (* R369 2 M DATA 삭제 완료 *)
    R369_2_M_NODE_4_09_통신_이상 AT %MW4524.9 : BOOL;
    R369_2_M_SEQ AT %MW10080 : WORD; (* R369 2 M SEQ *)
    R369_2_M_VIN_NO_1_2 AT %MW10091 : WORD; (* R369 2 M VIN NO 1 2 *)
    R369_2_M_VIN_NO_3_4 AT %MW10092 : WORD; (* R369 2 M VIN NO 3 4 *)
    R369_2_M_VIN_NO_5_6 AT %MW10093 : WORD; (* R369 2 M VIN NO 5 6 *)
    R369_2_M_VIN_NO_7_8 AT %MW10094 : WORD; (* R369 2 M VIN NO 7 8 *)
    R369_2_M_VIN_NO_9_10 AT %MW10095 : WORD; (* R369 2 M VIN NO 9 10 *)
    R369_2_M_로딩버퍼_DATA_전송_MEMO AT %MW9008.8 : BOOL; (* R369 2 M 로딩버퍼 DATA 전송 MEMO *)
    R369_2_M_로딩버퍼_DATA_전송_PLS AT %MW9008.9 : BOOL; (* R369 2 M 로딩버퍼 DATA 전송 PLS *)
    R369_2_M_로딩버퍼_DATA_전송_SIGN AT %MW9008.10 : BOOL; (* R369 2 M 로딩버퍼 DATA 전송 SIGN *)
    R369_2_M_로딩버퍼_DATA_전송_완료 AT %MW9008.11 : BOOL; (* R369 2 M 로딩버퍼 DATA 전송 완료 *)
    R369_2_M_차종1_AX AT %MW10081.0 : BOOL; (* R369 2 M 차종1 AX *)
    R369_2_M_차종1_B AT %MW10081.1 : BOOL; (* R369 2 M 차종1 B *)
    R369_2_M_차종1_C AT %MW10081.2 : BOOL; (* R369 2 M 차종1 C *)
    R369_2_M_차종1_D AT %MW10081.3 : BOOL; (* R369 2 M 차종1 D *)
    R369_2_M_차종1_E AT %MW10081.4 : BOOL; (* R369 2 M 차종1 E *)
    R369_2_M_차종1_F AT %MW10081.5 : BOOL; (* R369 2 M 차종1 F *)
    R369_2_M_차종1_G AT %MW10081.6 : BOOL; (* R369 2 M 차종1 G *)
    R369_2_M_차종1_H AT %MW10081.7 : BOOL; (* R369 2 M 차종1 H *)
    R369_2_M_차종2_3DR AT %MW10081.8 : BOOL; (* R369 2 M 차종2 3DR *)
    R369_2_M_차종2_4DR AT %MW10081.9 : BOOL; (* R369 2 M 차종2 4DR *)
    R369_2_M_차종2_5DR AT %MW10081.10 : BOOL; (* R369 2 M 차종2 5DR *)
    R369_2_M_차종2_SP1 AT %MW10081.12 : BOOL; (* R369 2 M 차종2 SP1 *)
    R369_2_M_차종2_SP2 AT %MW10081.13 : BOOL; (* R369 2 M 차종2 SP2 *)
    R369_2_M_차종2_WGN AT %MW10081.11 : BOOL; (* R369 2 M 차종2 WGN *)
    R369_2_M_차종3_LHD AT %MW10081.14 : BOOL; (* R369 2 M 차종3 LHD *)
    R369_2_M_차종3_RHD AT %MW10081.15 : BOOL; (* R369 2 M 차종3 RHD *)
    R369_2_M_차종4_EEC AT %MW10082.3 : BOOL; (* R369 2 M 차종4 EEC *)
    R369_2_M_차종4_SP1 AT %MW10082.8 : BOOL; (* R369 2 M 차종4 SP1 *)
    R369_2_M_차종4_SP2 AT %MW10082.9 : BOOL; (* R369 2 M 차종4 SP2 *)
    R369_2_M_차종4_SP3 AT %MW10082.11 : BOOL; (* R369 2 M 차종4 SP3 *)
    R369_2_M_차종4_SP4 AT %MW10082.12 : BOOL; (* R369 2 M 차종4 SP4 *)
    R369_2_M_차종4_SP5 AT %MW10082.13 : BOOL; (* R369 2 M 차종4 SP5 *)
    R369_2_M_차종4_SP6 AT %MW10082.14 : BOOL; (* R369 2 M 차종4 SP6 *)
    R369_2_M_차종4_SP7 AT %MW10082.15 : BOOL; (* R369 2 M 차종4 SP7 *)
    R369_2_M_차종4_내수 AT %MW10082.0 : BOOL; (* R369 2 M 차종4 내수 *)
    R369_2_M_차종4_러시아 AT %MW10082.10 : BOOL; (* R369 2 M 차종4 러시아 *)
    R369_2_M_차종4_북미 AT %MW10082.2 : BOOL; (* R369 2 M 차종4 북미 *)
    R369_2_M_차종4_브라질 AT %MW10082.7 : BOOL; (* R369 2 M 차종4 브라질 *)
    R369_2_M_차종4_수출 AT %MW10082.1 : BOOL; (* R369 2 M 차종4 수출 *)
    R369_2_M_차종4_중국 AT %MW10082.6 : BOOL; (* R369 2 M 차종4 중국 *)
    R369_2_M_차종4_중동 AT %MW10082.5 : BOOL; (* R369 2 M 차종4 중동 *)
    R369_2_M_차종4_호주 AT %MW10082.4 : BOOL; (* R369 2 M 차종4 호주 *)
    R369_2_M_차종5_AT AT %MW10083.1 : BOOL; (* R369 2 M 차종5 AT *)
    R369_2_M_차종5_MT AT %MW10083.0 : BOOL; (* R369 2 M 차종5 MT *)
    R369_2_M_차종5_SP1 AT %MW10083.2 : BOOL; (* R369 2 M 차종5 SP1 *)
    R369_2_M_차종6_DSROOF AT %MW10083.6 : BOOL; (* R369 2 M 차종6 DSROOF *)
    R369_2_M_차종6_SP1 AT %MW10083.7 : BOOL; (* R369 2 M 차종6 SP1 *)
    R369_2_M_차종6_썬루프 AT %MW10083.4 : BOOL; (* R369 2 M 차종6 썬루프 *)
    R369_2_M_차종6_일반루프 AT %MW10083.3 : BOOL; (* R369 2 M 차종6 일반루프 *)
    R369_2_M_차종6_파노라마루프 AT %MW10083.5 : BOOL; (* R369 2 M 차종6 파노라마루프 *)
    R369_2_M_차종7_DSL AT %MW10083.9 : BOOL; (* R369 2 M 차종7 DSL *)
    R369_2_M_차종7_GSL AT %MW10083.8 : BOOL; (* R369 2 M 차종7 GSL *)
    R369_2_M_차종7_SP1 AT %MW10083.10 : BOOL; (* R369 2 M 차종7 SP1 *)
    R369_2_M_차종7_SP2 AT %MW10083.11 : BOOL; (* R369 2 M 차종7 SP2 *)
    R369_2_M_차종7_SP3 AT %MW10083.12 : BOOL; (* R369 2 M 차종7 SP3 *)
    R369_2_M_차종7_SP4 AT %MW10083.13 : BOOL; (* R369 2 M 차종7 SP4 *)
    R369_2_M_차종7_SP5 AT %MW10083.14 : BOOL; (* R369 2 M 차종7 SP5 *)
    R369_2_M_차종7_SP6 AT %MW10083.15 : BOOL; (* R369 2 M 차종7 SP6 *)
    R369_2_M_차종8_2WD AT %MW10084.0 : BOOL; (* R369 2 M 차종8 2WD *)
    R369_2_M_차종8_4WD AT %MW10084.1 : BOOL; (* R369 2 M 차종8 4WD *)
    R369_2_M_차종8_SP1 AT %MW10084.2 : BOOL; (* R369 2 M 차종8 SP1 *)
    R369_2_M_차종9_MPI AT %MW10084.3 : BOOL; (* R369 2 M 차종9 MPI *)
    R369_2_M_차종9_SP1 AT %MW10084.5 : BOOL; (* R369 2 M 차종9 SP1 *)
    R369_2_M_차종9_SP10 AT %MW10084.14 : BOOL; (* R369 2 M 차종9 SP10 *)
    R369_2_M_차종9_SP11 AT %MW10084.15 : BOOL; (* R369 2 M 차종9 SP11 *)
    R369_2_M_차종9_SP2 AT %MW10084.6 : BOOL; (* R369 2 M 차종9 SP2 *)
    R369_2_M_차종9_SP3 AT %MW10084.7 : BOOL; (* R369 2 M 차종9 SP3 *)
    R369_2_M_차종9_SP4 AT %MW10084.8 : BOOL; (* R369 2 M 차종9 SP4 *)
    R369_2_M_차종9_SP5 AT %MW10084.9 : BOOL; (* R369 2 M 차종9 SP5 *)
    R369_2_M_차종9_SP6 AT %MW10084.10 : BOOL; (* R369 2 M 차종9 SP6 *)
    R369_2_M_차종9_SP7 AT %MW10084.11 : BOOL; (* R369 2 M 차종9 SP7 *)
    R369_2_M_차종9_SP8 AT %MW10084.12 : BOOL; (* R369 2 M 차종9 SP8 *)
    R369_2_M_차종9_SP9 AT %MW10084.13 : BOOL; (* R369 2 M 차종9 SP9 *)
    R369_2_M_차종9_T_GDI AT %MW10084.4 : BOOL; (* R369 2 M 차종9 T GDI *)
    R369_2_M_차종_AS AT %MW10090.9 : BOOL; (* R369 2 M 차종 AS *)
    R369_2_M_차종_OPT1_R_RACK_무 AT %MW10085.3 : BOOL; (* R369 2 M 차종 OPT1 R RACK 무 *)
    R369_2_M_차종_OPT1_R_RACK_유 AT %MW10085.2 : BOOL; (* R369 2 M 차종 OPT1 R RACK 유 *)
    R369_2_M_차종_OPT1_SP1 AT %MW10085.10 : BOOL; (* R369 2 M 차종 OPT1 SP1 *)
    R369_2_M_차종_OPT1_SP2 AT %MW10085.11 : BOOL; (* R369 2 M 차종 OPT1 SP2 *)
    R369_2_M_차종_OPT1_SP3 AT %MW10085.12 : BOOL; (* R369 2 M 차종 OPT1 SP3 *)
    R369_2_M_차종_OPT1_SP4 AT %MW10085.13 : BOOL; (* R369 2 M 차종 OPT1 SP4 *)
    R369_2_M_차종_OPT1_SP5 AT %MW10085.14 : BOOL; (* R369 2 M 차종 OPT1 SP5 *)
    R369_2_M_차종_OPT1_SP6 AT %MW10085.15 : BOOL; (* R369 2 M 차종 OPT1 SP6 *)
    R369_2_M_차종_OPT1_S_REP_EATER_무 AT %MW10085.7 : BOOL; (* R369 2 M 차종 OPT1 S REP EATER 무 *)
    R369_2_M_차종_OPT1_S_REP_EATER_유 AT %MW10085.6 : BOOL; (* R369 2 M 차종 OPT1 S REP EATER 유 *)
    R369_2_M_차종_OPT1_VAN_무 AT %MW10085.9 : BOOL; (* R369 2 M 차종 OPT1 VAN 무 *)
    R369_2_M_차종_OPT1_VAN_유 AT %MW10085.8 : BOOL; (* R369 2 M 차종 OPT1 VAN 유 *)
    R369_2_M_차종_OPT1_슬라이딩_무 AT %MW10085.1 : BOOL; (* R369 2 M 차종 OPT1 슬라이딩 무 *)
    R369_2_M_차종_OPT1_슬라이딩_유 AT %MW10085.0 : BOOL; (* R369 2 M 차종 OPT1 슬라이딩 유 *)
    R369_2_M_차종_OPT1_폴딩_무 AT %MW10085.5 : BOOL; (* R369 2 M 차종 OPT1 폴딩 무 *)
    R369_2_M_차종_OPT1_폴딩_유 AT %MW10085.4 : BOOL; (* R369 2 M 차종 OPT1 폴딩 유 *)
    R369_2_M_차종_OPT2_SP_WORD1 AT %MW10086 : WORD; (* R369 2 M 차종 OPT2 SP WORD1 *)
    R369_2_M_차종_OPT3_SP_WORD2 AT %MW10087 : WORD; (* R369 2 M 차종 OPT3 SP WORD2 *)
    R369_2_M_차종_OPT4_SP_WORD3 AT %MW10088 : WORD; (* R369 2 M 차종 OPT4 SP WORD3 *)
    R369_2_M_차종_OPT5_SP_WORD4 AT %MW10089 : WORD; (* R369 2 M 차종 OPT5 SP WORD4 *)
    R369_2_M_차종_SP1 AT %MW10090.0 : BOOL; (* R369 2 M 차종 SP1 *)
    R369_2_M_차종_SP2 AT %MW10090.1 : BOOL; (* R369 2 M 차종 SP2 *)
    R369_2_M_차종_SP3 AT %MW10090.2 : BOOL; (* R369 2 M 차종 SP3 *)
    R369_2_M_차종_SP4 AT %MW10090.3 : BOOL; (* R369 2 M 차종 SP4 *)
    R369_2_M_차종_SP5 AT %MW10090.4 : BOOL; (* R369 2 M 차종 SP5 *)
    R369_2_M_차종_SP6 AT %MW10090.5 : BOOL; (* R369 2 M 차종 SP6 *)
    R369_2_M_차종_SP7 AT %MW10090.6 : BOOL; (* R369 2 M 차종 SP7 *)
    R369_2_M_차종_SP8 AT %MW10090.7 : BOOL; (* R369 2 M 차종 SP8 *)
    R369_2_M_차종_SP9 AT %MW10090.15 : BOOL; (* R369 2 M 차종 SP9 *)
    R369_2_M_차종_공대차 AT %MW10090.12 : BOOL; (* R369 2 M 차종 공대차 *)
    R369_2_M_차종_공차 AT %MW10090.10 : BOOL; (* R369 2 M 차종 공차 *)
    R369_2_M_차종_무 AT %MW4502.5 : BOOL;
    R369_2_M_차종_불량대차 AT %MW10090.13 : BOOL; (* R369 2 M 차종 불량대차 *)
    R369_2_M_차종_불량차 AT %MW10090.11 : BOOL; (* R369 2 M 차종 불량차 *)
    R369_2_M_차종_비축 AT %MW10090.8 : BOOL; (* R369 2 M 차종 비축 *)
    R369_2_M_차종_유 AT %MW4502.4 : BOOL;
    R369_2_M_차종_취출대차 AT %MW10090.14 : BOOL; (* R369 2 M 차종 취출대차 *)
    ROOF_RACK1_3_M_NODE_7_40_통신_이상 AT %MW1524.0 : BOOL;
    ROOF_RACK1_M_HMI입력_차종 AT %MW501 : WORD;
    ROOF_RACK1_M_LC_이상 AT %MW1512.0 : BOOL;
    ROOF_RACK1_M_LC_정상 AT %MW1505.0 : BOOL;
    ROOF_RACK1_M_PLT_이상 AT %MW1514.0 : BOOL;
    ROOF_RACK1_M_랙감지_무 AT %MW1501.1 : BOOL;
    ROOF_RACK1_M_랙감지_유 AT %MW1501.0 : BOOL;
    ROOF_RACK1_M_로딩완료 AT %MW1561.0 : BOOL;
    ROOF_RACK1_M_막장감지_무 AT %MW1503.1 : BOOL;
    ROOF_RACK1_M_막장감지_유 AT %MW1503.0 : BOOL;
    ROOF_RACK1_M_발목감지_이상 AT %MW1512.8 : BOOL;
    ROOF_RACK1_M_발목감지_정상 AT %MW1506.0 : BOOL;
    ROOF_RACK1_M_우선순위_지정 AT %MW1564.0 : BOOL;
    ROOF_RACK1_M_제품수량 AT %MW511 : WORD;
    ROOF_RACK1_M_차종 AT %MW1541 : WORD;
    ROOF_RACK1_M_차종_무 AT %MW1540.1 : BOOL;
    ROOF_RACK1_M_차종_유 AT %MW1540.0 : BOOL;
    ROOF_RACK1_M_차종_이상 AT %MW1515.0 : BOOL;
    ROOF_RACK1_M_카운트_리셋요구_SET AT %MW1566.0 : BOOL;
    ROOF_RACK2_M_HMI입력_차종 AT %MW502 : WORD;
    ROOF_RACK2_M_LC_이상 AT %MW1512.1 : BOOL;
    ROOF_RACK2_M_LC_정상 AT %MW1505.1 : BOOL;
    ROOF_RACK2_M_PLT_이상 AT %MW1514.1 : BOOL;
    ROOF_RACK2_M_랙감지_무 AT %MW1501.3 : BOOL;
    ROOF_RACK2_M_랙감지_유 AT %MW1501.2 : BOOL;
    ROOF_RACK2_M_로딩완료 AT %MW1561.1 : BOOL;
    ROOF_RACK2_M_막장감지_무 AT %MW1503.3 : BOOL;
    ROOF_RACK2_M_막장감지_유 AT %MW1503.2 : BOOL;
    ROOF_RACK2_M_발목감지_이상 AT %MW1512.9 : BOOL;
    ROOF_RACK2_M_발목감지_정상 AT %MW1506.1 : BOOL;
    ROOF_RACK2_M_우선순위_지정 AT %MW1564.1 : BOOL;
    ROOF_RACK2_M_제품수량 AT %MW512 : WORD;
    ROOF_RACK2_M_차종 AT %MW1542 : WORD;
    ROOF_RACK2_M_차종_무 AT %MW1540.3 : BOOL;
    ROOF_RACK2_M_차종_유 AT %MW1540.2 : BOOL;
    ROOF_RACK2_M_차종_이상 AT %MW1515.1 : BOOL;
    ROOF_RACK2_M_카운트_리셋요구_SET AT %MW1566.1 : BOOL;
    ROOF_RACK3_M_HMI입력_차종 AT %MW503 : WORD;
    ROOF_RACK3_M_LC_이상 AT %MW1512.2 : BOOL;
    ROOF_RACK3_M_LC_정상 AT %MW1505.2 : BOOL;
    ROOF_RACK3_M_PLT_이상 AT %MW1514.2 : BOOL;
    ROOF_RACK3_M_랙감지_무 AT %MW1501.5 : BOOL;
    ROOF_RACK3_M_랙감지_유 AT %MW1501.4 : BOOL;
    ROOF_RACK3_M_로딩완료 AT %MW1561.2 : BOOL;
    ROOF_RACK3_M_막장감지_무 AT %MW1503.5 : BOOL;
    ROOF_RACK3_M_막장감지_유 AT %MW1503.4 : BOOL;
    ROOF_RACK3_M_발목감지_이상 AT %MW1512.10 : BOOL;
    ROOF_RACK3_M_발목감지_정상 AT %MW1506.2 : BOOL;
    ROOF_RACK3_M_우선순위_지정 AT %MW1564.2 : BOOL;
    ROOF_RACK3_M_제품수량 AT %MW513 : WORD;
    ROOF_RACK3_M_차종 AT %MW1543 : WORD;
    ROOF_RACK3_M_차종_무 AT %MW1540.5 : BOOL;
    ROOF_RACK3_M_차종_유 AT %MW1540.4 : BOOL;
    ROOF_RACK3_M_차종_이상 AT %MW1515.2 : BOOL;
    ROOF_RACK3_M_카운트_리셋요구_SET AT %MW1566.2 : BOOL;
    ROOF_RACK4_6_M_NODE_7_45_통신_이상 AT %MW1524.1 : BOOL;
    ROOF_RACK4_M_HMI입력_차종 AT %MW504 : WORD;
    ROOF_RACK4_M_LC_이상 AT %MW1512.3 : BOOL;
    ROOF_RACK4_M_LC_정상 AT %MW1505.3 : BOOL;
    ROOF_RACK4_M_PLT_이상 AT %MW1514.3 : BOOL;
    ROOF_RACK4_M_랙감지_무 AT %MW1501.7 : BOOL;
    ROOF_RACK4_M_랙감지_유 AT %MW1501.6 : BOOL;
    ROOF_RACK4_M_로딩완료 AT %MW1561.3 : BOOL;
    ROOF_RACK4_M_막장감지_무 AT %MW1503.7 : BOOL;
    ROOF_RACK4_M_막장감지_유 AT %MW1503.6 : BOOL;
    ROOF_RACK4_M_발목감지_이상 AT %MW1512.11 : BOOL;
    ROOF_RACK4_M_발목감지_정상 AT %MW1506.3 : BOOL;
    ROOF_RACK4_M_우선순위_지정 AT %MW1564.3 : BOOL;
    ROOF_RACK4_M_제품수량 AT %MW514 : WORD;
    ROOF_RACK4_M_차종 AT %MW1544 : WORD;
    ROOF_RACK4_M_차종_무 AT %MW1540.7 : BOOL;
    ROOF_RACK4_M_차종_유 AT %MW1540.6 : BOOL;
    ROOF_RACK4_M_차종_이상 AT %MW1515.3 : BOOL;
    ROOF_RACK4_M_카운트_리셋요구_SET AT %MW1566.3 : BOOL;
    ROOF_RACK5_M_HMI입력_차종 AT %MW505 : WORD;
    ROOF_RACK5_M_LC_이상 AT %MW1512.4 : BOOL;
    ROOF_RACK5_M_LC_정상 AT %MW1505.4 : BOOL;
    ROOF_RACK5_M_PLT_이상 AT %MW1514.4 : BOOL;
    ROOF_RACK5_M_랙감지_무 AT %MW1501.9 : BOOL;
    ROOF_RACK5_M_랙감지_유 AT %MW1501.8 : BOOL;
    ROOF_RACK5_M_로딩완료 AT %MW1561.4 : BOOL;
    ROOF_RACK5_M_막장감지_무 AT %MW1503.9 : BOOL;
    ROOF_RACK5_M_막장감지_유 AT %MW1503.8 : BOOL;
    ROOF_RACK5_M_발목감지_이상 AT %MW1512.12 : BOOL;
    ROOF_RACK5_M_발목감지_정상 AT %MW1506.4 : BOOL;
    ROOF_RACK5_M_우선순위_지정 AT %MW1564.4 : BOOL;
    ROOF_RACK5_M_제품수량 AT %MW515 : WORD;
    ROOF_RACK5_M_차종 AT %MW1545 : WORD;
    ROOF_RACK5_M_차종_무 AT %MW1540.9 : BOOL;
    ROOF_RACK5_M_차종_유 AT %MW1540.8 : BOOL;
    ROOF_RACK5_M_차종_이상 AT %MW1515.4 : BOOL;
    ROOF_RACK5_M_카운트_리셋요구_SET AT %MW1566.4 : BOOL;
    ROOF_RACK6_M_HMI입력_차종 AT %MW506 : WORD;
    ROOF_RACK6_M_LC_이상 AT %MW1512.5 : BOOL;
    ROOF_RACK6_M_LC_정상 AT %MW1505.5 : BOOL;
    ROOF_RACK6_M_PLT_이상 AT %MW1514.5 : BOOL;
    ROOF_RACK6_M_랙감지_무 AT %MW1501.11 : BOOL;
    ROOF_RACK6_M_랙감지_유 AT %MW1501.10 : BOOL;
    ROOF_RACK6_M_로딩완료 AT %MW1561.5 : BOOL;
    ROOF_RACK6_M_막장감지_무 AT %MW1503.11 : BOOL;
    ROOF_RACK6_M_막장감지_유 AT %MW1503.10 : BOOL;
    ROOF_RACK6_M_발목감지_이상 AT %MW1512.13 : BOOL;
    ROOF_RACK6_M_발목감지_정상 AT %MW1506.5 : BOOL;
    ROOF_RACK6_M_우선순위_지정 AT %MW1564.5 : BOOL;
    ROOF_RACK6_M_제품수량 AT %MW516 : WORD;
    ROOF_RACK6_M_차종 AT %MW1546 : WORD;
    ROOF_RACK6_M_차종_무 AT %MW1540.11 : BOOL;
    ROOF_RACK6_M_차종_유 AT %MW1540.10 : BOOL;
    ROOF_RACK6_M_차종_이상 AT %MW1515.5 : BOOL;
    ROOF_RACK6_M_카운트_리셋요구_SET AT %MW1566.5 : BOOL;
    ROOF_RACK_1_3_M_CP_이상 AT %MW1517.0 : BOOL;
    ROOF_RACK_4_6_M_CP_이상 AT %MW1517.1 : BOOL;
    ROOF_RACK_M_RB_ESTOP_NORMAL AT %MW1504.0 : BOOL;
    ROOF_RACK_M_버퍼1_지정 AT %MW1562.0 : BOOL;
    ROOF_RACK_M_버퍼2_지정 AT %MW1562.1 : BOOL;
    ROOF_RACK_M_버퍼3_지정 AT %MW1562.2 : BOOL;
    ROOF_RACK_M_버퍼4_지정 AT %MW1562.3 : BOOL;
    ROOF_RACK_M_버퍼5_지정 AT %MW1562.4 : BOOL;
    ROOF_RACK_M_버퍼6_지정 AT %MW1562.5 : BOOL;
    ROOF_RACK_M_수동모드 AT %MW1500.3 : BOOL;
    ROOF_RACK_M_우선순위_버퍼1 AT %MW1551 : WORD;
    ROOF_RACK_M_우선순위_버퍼2 AT %MW1552 : WORD;
    ROOF_RACK_M_우선순위_버퍼3 AT %MW1553 : WORD;
    ROOF_RACK_M_우선순위_버퍼4 AT %MW1554 : WORD;
    ROOF_RACK_M_우선순위_버퍼5 AT %MW1555 : WORD;
    ROOF_RACK_M_우선순위_버퍼6 AT %MW1556 : WORD;
    ROOF_RACK_M_운전준비_ON AT %MW1500.0 : BOOL;
    ROOF_RACK_M_자동_START AT %MW1500.5 : BOOL;
    ROOF_RACK_M_자동_운전중 AT %MW1500.4 : BOOL;
    ROOF_RACK_M_자동모드 AT %MW1500.1 : BOOL;
    ROOF_RACK_M_작업완료_SET_PLS AT %MW1500.8 : BOOL;
    ROOF_RACK_M_작업완료_리셋_PLS AT %MW1500.9 : BOOL;
    ROOF_RACK_M_전체_LC_정상 AT %MW1504.4 : BOOL;
    ROOF_RACK_M_전체_SAFETY_정상 AT %MW1504.2 : BOOL;
    ROOF_RACK_M_전체_발목감지_정상 AT %MW1504.6 : BOOL;
    ROOF_RACK_M_총괄_CP_이상 AT %MW1509.7 : BOOL;
    ROOF_RACK_M_총괄_CT_이상 AT %MW1510.4 : BOOL;
    ROOF_RACK_M_총괄_EOCR_이상 AT %MW1509.8 : BOOL;
    ROOF_RACK_M_총괄_INV_이상 AT %MW1509.9 : BOOL;
    ROOF_RACK_M_총괄_LS_이상 AT %MW1509.15 : BOOL;
    ROOF_RACK_M_총괄_MATCH_이상 AT %MW1510.0 : BOOL;
    ROOF_RACK_M_총괄_MC_이상 AT %MW1509.13 : BOOL;
    ROOF_RACK_M_총괄_MOTOR_이상 AT %MW1510.3 : BOOL;
    ROOF_RACK_M_총괄_NFB_이상 AT %MW1509.11 : BOOL;
    ROOF_RACK_M_총괄_ROBOT_이상 AT %MW1510.1 : BOOL;
    ROOF_RACK_M_총괄_SAFETY_이상 AT %MW1509.2 : BOOL;
    ROOF_RACK_M_총괄_SRV_이상 AT %MW1509.10 : BOOL;
    ROOF_RACK_M_총괄_공기압_이상 AT %MW1509.3 : BOOL;
    ROOF_RACK_M_총괄_비상정지_이상 AT %MW1509.1 : BOOL;
    ROOF_RACK_M_총괄_사양_이상 AT %MW1509.6 : BOOL;
    ROOF_RACK_M_총괄_오버런_이상 AT %MW1509.12 : BOOL;
    ROOF_RACK_M_총괄_용접타점수_이상 AT %MW1510.2 : BOOL;
    ROOF_RACK_M_총괄_이상 AT %MW1509.0 : BOOL;
    ROOF_RACK_M_총괄_제품감지_이상 AT %MW1509.4 : BOOL;
    ROOF_RACK_M_총괄_차종_이상 AT %MW1509.5 : BOOL;
    ROOF_RACK_M_총괄_통신_이상 AT %MW1509.14 : BOOL;
    S163_M_LH_TURN_LS_이상 AT %MW4100.7 : BOOL; (* S163_M_LH_TURN_LS_이상 *)
    S301_M_자동_운전중 : BOOL; (* S301 M 자동 운전중 *)
    S362_HOME AT %MW1048.0 : BOOL; (* S362_HOME *)
    S362_M_AOP_비상정지_이상 AT %MW1011.0 : BOOL; (* S362_M_AOP_비상정지_이상 *)
    S362_M_BYPASS_보조 AT %MW1003.15 : BOOL; (* S362 M BYPASS 보조 *)
    S362_M_CTIME_OVER_ALRAM AT %MW1007.14 : BOOL; (* S362_M_CTIME_OVER_ALRAM *)
    S362_M_CTIME_OVER_MUTE AT %MW1007.13 : BOOL; (* S362_M_CTIME_OVER_MUTE *)
    S362_M_DATA_삭제_PLS AT %MW9010.0 : BOOL; (* S362 M DATA 삭제 PLS *)
    S362_M_DATA_삭제_SIGN AT %MW9010.1 : BOOL; (* S362 M DATA 삭제 SIGN *)
    S362_M_DATA_삭제_완료 AT %MW9010.2 : BOOL; (* S362 M DATA 삭제 완료 *)
    S362_M_LC_정상 AT %MW1007.5 : BOOL; (* S362_M_LC_정상 *)
    S362_M_LH_CB_OFF AT %MW1021.1 : BOOL; (* S362_M_LH_CB_OFF *)
    S362_M_LH_INV_이상 AT %MW1019.0 : BOOL; (* S362_M_LH_INV_이상 *)
    S362_M_LH_MC_이상 AT %MW1023.0 : BOOL; (* S362_M_LH_MC_이상 *)
    S362_M_LH_NFB_OFF AT %MW1021.0 : BOOL; (* S362_M_LH_NFB_OFF *)
    S362_M_LH_STEP_MOVE_리셋_PLS AT %MW1104.14 : BOOL; (* S362_M_LH_STEP_MOVE_리셋_PLS *)
    S362_M_LH_TURN_1_포지션단 AT %MW1104.3 : BOOL; (* S362_M_LH_TURN_1_포지션단 *)
    S362_M_LH_TURN_2_포지션단 AT %MW1104.4 : BOOL; (* S362_M_LH_TURN_2_포지션단 *)
    S362_M_LH_TURN_3_포지션단 AT %MW1104.5 : BOOL; (* S362_M_LH_TURN_3_포지션단 *)
    S362_M_LH_TURN_4_포지션단 AT %MW1104.6 : BOOL; (* S362_M_LH_TURN_4_포지션단 *)
    S362_M_LH_TURN_LS_이상 AT %MW1104.7 : BOOL; (* S362_M_LH_TURN_LS_이상 *)
    S362_M_LH_TURN_MOVE_완료 AT %MW1104.8 : BOOL; (* S362_M_LH_TURN_MOVE_완료 *)
    S362_M_LH_TURN_수동_STEP_전진_보조 AT %MW1104.11 : BOOL; (* S362_M_LH_TURN_수동_STEP_전진_보조 *)
    S362_M_LH_TURN_수동_STEP_후진_보조 AT %MW1104.12 : BOOL; (* S362_M_LH_TURN_수동_STEP_후진_보조 *)
    S362_M_LH_TURN_수동_전진_보조 AT %MW1104.9 : BOOL; (* S362_M_LH_TURN_수동_전진_보조 *)
    S362_M_LH_TURN_수동_후진_보조 AT %MW1104.10 : BOOL; (* S362_M_LH_TURN_수동_후진_보조 *)
    S362_M_LH_TURN_전진_보조 AT %MW1104.1 : BOOL; (* S362_M_LH_TURN_전진_보조 *)
    S362_M_LH_TURN_조건 AT %MW1104.0 : BOOL; (* S362_M_LH_TURN_조건 *)
    S362_M_LH_TURN_후진_보조 AT %MW1104.2 : BOOL; (* S362_M_LH_TURN_후진_보조 *)
    S362_M_LH_자동_MOVE_리셋_PLS AT %MW1104.13 : BOOL; (* S362_M_LH_자동_MOVE_리셋_PLS *)
    S362_M_MAT_정상 AT %MW1007.6 : BOOL; (* S362_M_MAT_정상 *)
    S362_M_NODE_7_10_통신_이상 AT %MW1024.0 : BOOL;
    S362_M_OP_ESTOP_NORMAL AT %MW1007.1 : BOOL; (* S362_M_OP_ESTOP_NORMAL *)
    S362_M_OP_LC_이상 AT %MW1012.0 : BOOL; (* S362_M_OP_LC_이상 *)
    S362_M_OP_MAT_이상 AT %MW1012.1 : BOOL; (* S362_M_OP_MAT_이상 *)
    S362_M_R363_1_실링완료 AT %MW1001.2 : BOOL;
    S362_M_R363_2_DATA_전송_MEMO AT %MW9010.4 : BOOL; (* S362 M R363 2 DATA 전송 MEMO *)
    S362_M_R363_2_DATA_전송_PLS AT %MW9010.5 : BOOL; (* S362 M R363 2 DATA 전송 PLS *)
    S362_M_R363_2_DATA_전송_SIGN AT %MW9010.6 : BOOL; (* S362 M R363 2 DATA 전송 SIGN *)
    S362_M_R363_2_DATA_전송_완료 AT %MW9010.7 : BOOL; (* S362 M R363 2 DATA 전송 완료 *)
    S362_M_R363_2_언로딩_완료 AT %MW1001.3 : BOOL;
    S362_M_RH_CB_OFF AT %MW1021.4 : BOOL; (* S362_M_RH_CB_OFF *)
    S362_M_RH_INV_이상 AT %MW1019.1 : BOOL; (* S362_M_RH_INV_이상 *)
    S362_M_RH_MC_이상 AT %MW1023.1 : BOOL; (* S362_M_RH_MC_이상 *)
    S362_M_RH_NFB_OFF AT %MW1021.3 : BOOL; (* S362_M_RH_NFB_OFF *)
    S362_M_RH_STEP_MOVE_리셋_PLS AT %MW1112.14 : BOOL; (* S362_M_RH_STEP_MOVE_리셋_PLS *)
    S362_M_RH_TURN_1_포지션단 AT %MW1112.3 : BOOL; (* S362_M_RH_TURN_1_포지션단 *)
    S362_M_RH_TURN_2_포지션단 AT %MW1112.4 : BOOL; (* S362_M_RH_TURN_2_포지션단 *)
    S362_M_RH_TURN_3_포지션단 AT %MW1112.5 : BOOL; (* S362_M_RH_TURN_3_포지션단 *)
    S362_M_RH_TURN_4_포지션단 AT %MW1112.6 : BOOL; (* S362_M_RH_TURN_4_포지션단 *)
    S362_M_RH_TURN_LS_이상 AT %MW1112.7 : BOOL; (* S362_M_RH_TURN_LS_이상 *)
    S362_M_RH_TURN_MOVE_완료 AT %MW1112.8 : BOOL; (* S362_M_RH_TURN_MOVE_완료 *)
    S362_M_RH_TURN_수동_STEP_전진_보조 AT %MW1112.11 : BOOL; (* S362_M_RH_TURN_수동_STEP_전진_보조 *)
    S362_M_RH_TURN_수동_STEP_후진_보조 AT %MW1112.12 : BOOL; (* S362_M_RH_TURN_수동_STEP_후진_보조 *)
    S362_M_RH_TURN_수동_전진_보조 AT %MW1112.9 : BOOL; (* S362_M_RH_TURN_수동_전진_보조 *)
    S362_M_RH_TURN_수동_후진_보조 AT %MW1112.10 : BOOL; (* S362_M_RH_TURN_수동_후진_보조 *)
    S362_M_RH_TURN_전진_보조 AT %MW1112.1 : BOOL; (* S362_M_RH_TURN_전진_보조 *)
    S362_M_RH_TURN_조건 AT %MW1112.0 : BOOL; (* S362_M_RH_TURN_조건 *)
    S362_M_RH_TURN_후진_보조 AT %MW1112.2 : BOOL; (* S362_M_RH_TURN_후진_보조 *)
    S362_M_RH_자동_MOVE_리셋_PLS AT %MW1112.13 : BOOL; (* S362_M_RH_자동_MOVE_리셋_PLS *)
    S362_M_S102_간섭무 AT %MW1004.2 : BOOL; (* S362_M_S102_간섭무 *)
    S362_M_SAFETY_불간섭 AT %MW1004.4 : BOOL; (* S362_M_SAFETY_불간섭 *)
    S362_M_SEMI_자동모드 AT %MW1000.2 : BOOL; (* S362_M_SEMI_자동모드 *)
    S362_M_SEQ AT %MW10100 : WORD; (* S362 M SEQ *)
    S362_M_SLD_LOCK_전진_LS_이상 AT %MW1102.5 : BOOL; (* S362_M_SLD_LOCK_전진_LS_이상 *)
    S362_M_SLD_LOCK_전진_보조 AT %MW1102.1 : BOOL; (* S362_M_SLD_LOCK_전진_보조 *)
    S362_M_SLD_LOCK_전진단 AT %MW1102.3 : BOOL; (* S362_M_SLD_LOCK_전진단 *)
    S362_M_SLD_LOCK_조건 AT %MW1102.0 : BOOL; (* S362_M_SLD_LOCK_조건 *)
    S362_M_SLD_LOCK_후진_LS_이상 AT %MW1102.6 : BOOL; (* S362_M_SLD_LOCK_후진_LS_이상 *)
    S362_M_SLD_LOCK_후진_보조 AT %MW1102.2 : BOOL; (* S362_M_SLD_LOCK_후진_보조 *)
    S362_M_SLD_LOCK_후진단 AT %MW1102.4 : BOOL; (* S362_M_SLD_LOCK_후진단 *)
    S362_M_SLIDE_전진_LS_이상 AT %MW1101.5 : BOOL; (* S362_M_SLIDE_전진_LS_이상 *)
    S362_M_SLIDE_전진_보조 AT %MW1101.1 : BOOL; (* S362_M_SLIDE_전진_보조 *)
    S362_M_SLIDE_전진단 AT %MW1101.3 : BOOL; (* S362_M_SLIDE_전진단 *)
    S362_M_SLIDE_조건 AT %MW1101.0 : BOOL; (* S362_M_SLIDE_조건 *)
    S362_M_SLIDE_후진_LS_이상 AT %MW1101.6 : BOOL; (* S362_M_SLIDE_후진_LS_이상 *)
    S362_M_SLIDE_후진_보조 AT %MW1101.2 : BOOL; (* S362_M_SLIDE_후진_보조 *)
    S362_M_SLIDE_후진단 AT %MW1101.4 : BOOL; (* S362_M_SLIDE_후진단 *)
    S362_M_TURN_LOCK_전진_LS_이상 AT %MW1100.5 : BOOL; (* S362_M_TURN_LOCK_전진_LS_이상 *)
    S362_M_TURN_LOCK_전진_보조 AT %MW1100.1 : BOOL; (* S362_M_TURN_LOCK_전진_보조 *)
    S362_M_TURN_LOCK_전진단 AT %MW1100.3 : BOOL; (* S362_M_TURN_LOCK_전진단 *)
    S362_M_TURN_LOCK_조건 AT %MW1100.0 : BOOL; (* S362_M_TURN_LOCK_조건 *)
    S362_M_TURN_LOCK_후진_LS_이상 AT %MW1100.6 : BOOL; (* S362_M_TURN_LOCK_후진_LS_이상 *)
    S362_M_TURN_LOCK_후진_보조 AT %MW1100.2 : BOOL; (* S362_M_TURN_LOCK_후진_보조 *)
    S362_M_TURN_LOCK_후진단 AT %MW1100.4 : BOOL; (* S362_M_TURN_LOCK_후진단 *)
    S362_M_VIN_NO_1_2 AT %MW10111 : WORD; (* S362 M VIN NO 1 2 *)
    S362_M_VIN_NO_3_4 AT %MW10112 : WORD; (* S362 M VIN NO 3 4 *)
    S362_M_VIN_NO_5_6 AT %MW10113 : WORD; (* S362 M VIN NO 5 6 *)
    S362_M_VIN_NO_7_8 AT %MW10114 : WORD; (* S362 M VIN NO 7 8 *)
    S362_M_VIN_NO_9_10 AT %MW10115 : WORD; (* S362 M VIN NO 9 10 *)
    S362_M_공정_AX_RAIL_제품감지_무 AT %MW1001.13 : BOOL; (* S362 M 공정 AX RAIL 제품감지 무 *)
    S362_M_공정_AX_RAIL_제품감지_유 AT %MW1001.12 : BOOL; (* S362 M 공정 AX RAIL 제품감지 유 *)
    S362_M_공정_AX_RAIL_제품감지_이상 AT %MW1014.3 : BOOL;
    S362_M_공정_AX_공용_제품감지_무 AT %MW1001.7 : BOOL; (* S362 M 공정 AX 공용 제품감지 무 *)
    S362_M_공정_AX_공용_제품감지_유 AT %MW1001.6 : BOOL; (* S362 M 공정 AX 공용 제품감지 유 *)
    S362_M_공정_AX_공용_제품감지_이상 AT %MW1014.0 : BOOL;
    S362_M_공정_AX_썬루프_제품감지_무 AT %MW1001.11 : BOOL; (* S362 M 공정 AX 썬루프 제품감지 무 *)
    S362_M_공정_AX_썬루프_제품감지_유 AT %MW1001.10 : BOOL; (* S362 M 공정 AX 썬루프 제품감지 유 *)
    S362_M_공정_AX_썬루프_제품감지_이상 AT %MW1014.2 : BOOL;
    S362_M_공정_AX_일반루프_제품감지_무 AT %MW1001.9 : BOOL; (* S362 M 공정 AX 일반루프 제품감지 무 *)
    S362_M_공정_AX_일반루프_제품감지_유 AT %MW1001.8 : BOOL; (* S362 M 공정 AX 일반루프 제품감지 유 *)
    S362_M_공정_AX_일반루프_제품감지_이상 AT %MW1014.1 : BOOL;
    S362_M_공정_SAFETY_NORMAL AT %MW1007.7 : BOOL; (* S362_M_공정_SAFETY_NORMAL *)
    S362_M_공정_불간섭 AT %MW1004.1 : BOOL; (* S362_M_공정_불간섭 *)
    S362_M_공정_원위치 AT %MW1004.0 : BOOL; (* S362_M_공정_원위치 *)
    S362_M_공정_제품감지_무 AT %MW1001.5 : BOOL; (* S362_M_공정_제품감지_무 *)
    S362_M_공정_제품감지_유 AT %MW1001.4 : BOOL; (* S362_M_공정_제품감지_유 *)
    S362_M_공정_차종_무 AT %MW1002.1 : BOOL; (* S362_M_공정_차종_무 *)
    S362_M_공정_차종_유 AT %MW1002.0 : BOOL; (* S362_M_공정_차종_유 *)
    S362_M_동작_선택_1 AT %MW1040.0 : BOOL; (* S362_M_동작_선택_1 *)
    S362_M_동작_선택_10 AT %MW1040.9 : BOOL; (* S362_M_동작_선택_10 *)
    S362_M_동작_선택_11 AT %MW1040.10 : BOOL; (* S362_M_동작_선택_11 *)
    S362_M_동작_선택_12 AT %MW1040.11 : BOOL; (* S362_M_동작_선택_12 *)
    S362_M_동작_선택_13 AT %MW1040.12 : BOOL; (* S362_M_동작_선택_13 *)
    S362_M_동작_선택_14 AT %MW1040.13 : BOOL; (* S362_M_동작_선택_14 *)
    S362_M_동작_선택_15 AT %MW1040.14 : BOOL; (* S362_M_동작_선택_15 *)
    S362_M_동작_선택_16 AT %MW1040.15 : BOOL; (* S362_M_동작_선택_16 *)
    S362_M_동작_선택_17 AT %MW1041.0 : BOOL; (* S362_M_동작_선택_17 *)
    S362_M_동작_선택_18 AT %MW1041.1 : BOOL; (* S362_M_동작_선택_18 *)
    S362_M_동작_선택_19 AT %MW1041.2 : BOOL; (* S362_M_동작_선택_19 *)
    S362_M_동작_선택_2 AT %MW1040.1 : BOOL; (* S362_M_동작_선택_2 *)
    S362_M_동작_선택_20 AT %MW1041.3 : BOOL; (* S362_M_동작_선택_20 *)
    S362_M_동작_선택_21 AT %MW1041.4 : BOOL; (* S362_M_동작_선택_21 *)
    S362_M_동작_선택_22 AT %MW1041.5 : BOOL; (* S362_M_동작_선택_22 *)
    S362_M_동작_선택_23 AT %MW1041.6 : BOOL; (* S362_M_동작_선택_23 *)
    S362_M_동작_선택_24 AT %MW1041.7 : BOOL; (* S362_M_동작_선택_24 *)
    S362_M_동작_선택_25 AT %MW1041.8 : BOOL; (* S362_M_동작_선택_25 *)
    S362_M_동작_선택_26 AT %MW1041.9 : BOOL; (* S362_M_동작_선택_26 *)
    S362_M_동작_선택_27 AT %MW1041.10 : BOOL; (* S362_M_동작_선택_27 *)
    S362_M_동작_선택_28 AT %MW1041.11 : BOOL; (* S362_M_동작_선택_28 *)
    S362_M_동작_선택_29 AT %MW1041.12 : BOOL; (* S362_M_동작_선택_29 *)
    S362_M_동작_선택_3 AT %MW1040.2 : BOOL; (* S362_M_동작_선택_3 *)
    S362_M_동작_선택_30 AT %MW1041.13 : BOOL; (* S362_M_동작_선택_30 *)
    S362_M_동작_선택_31 AT %MW1041.14 : BOOL; (* S362_M_동작_선택_31 *)
    S362_M_동작_선택_32 AT %MW1041.15 : BOOL; (* S362_M_동작_선택_32 *)
    S362_M_동작_선택_4 AT %MW1040.3 : BOOL; (* S362_M_동작_선택_4 *)
    S362_M_동작_선택_5 AT %MW1040.4 : BOOL; (* S362_M_동작_선택_5 *)
    S362_M_동작_선택_6 AT %MW1040.5 : BOOL; (* S362_M_동작_선택_6 *)
    S362_M_동작_선택_7 AT %MW1040.6 : BOOL; (* S362_M_동작_선택_7 *)
    S362_M_동작_선택_8 AT %MW1040.7 : BOOL; (* S362_M_동작_선택_8 *)
    S362_M_동작_선택_9 AT %MW1040.8 : BOOL; (* S362_M_동작_선택_9 *)
    S362_M_부저_정지_보조 AT %MW1000.11 : BOOL; (* S362_M_부저_정지_보조 *)
    S362_M_수동모드 AT %MW1000.3 : BOOL; (* S362 선택 수동모드 *)
    S362_M_썬루프_사양_이상 AT %MW1016.1 : BOOL;
    S362_M_운전준비_ON AT %MW1000.0 : BOOL; (* S362 운전준비 ON *)
    S362_M_이상_리셋_보조 AT %MW1000.10 : BOOL; (* S362_M_이상_리셋_보조 *)
    S362_M_일반루프_사양_이상 AT %MW1016.0 : BOOL;
    S362_M_자동_START AT %MW1000.5 : BOOL; (* S362 자동운전중 *)
    S362_M_자동_운전중 AT %MW1000.4 : BOOL; (* S362 자동운전중 *)
    S362_M_자동모드 AT %MW1000.1 : BOOL; (* S362 선택 자동모드 *)
    S362_M_작업_완료 AT %MW1001.0 : BOOL; (* S362_M_작업_완료 *)
    S362_M_작업완료_SET_PLS AT %MW1000.8 : BOOL; (* S362 M 작업완료 SET PLS *)
    S362_M_작업완료_리셋_PLS AT %MW1000.9 : BOOL; (* S362 M 작업완료 리셋 PLS *)
    S362_M_작업자_작업_가능 AT %MW1004.8 : BOOL; (* S362 M 작업자 작업 가능 *)
    S362_M_작업자_작업완료 AT %MW1001.1 : BOOL;
    S362_M_차종1_AX AT %MW10101.0 : BOOL; (* S362 M 차종1 AX *)
    S362_M_차종1_B AT %MW10101.1 : BOOL; (* S362 M 차종1 B *)
    S362_M_차종1_C AT %MW10101.2 : BOOL; (* S362 M 차종1 C *)
    S362_M_차종1_D AT %MW10101.3 : BOOL; (* S362 M 차종1 D *)
    S362_M_차종1_E AT %MW10101.4 : BOOL; (* S362 M 차종1 E *)
    S362_M_차종1_F AT %MW10101.5 : BOOL; (* S362 M 차종1 F *)
    S362_M_차종1_G AT %MW10101.6 : BOOL; (* S362 M 차종1 G *)
    S362_M_차종1_H AT %MW10101.7 : BOOL; (* S362 M 차종1 H *)
    S362_M_차종2_3DR AT %MW10101.8 : BOOL; (* S362 M 차종2 3DR *)
    S362_M_차종2_4DR AT %MW10101.9 : BOOL; (* S362 M 차종2 4DR *)
    S362_M_차종2_5DR AT %MW10101.10 : BOOL; (* S362 M 차종2 5DR *)
    S362_M_차종2_SP1 AT %MW10101.12 : BOOL; (* S362 M 차종2 SP1 *)
    S362_M_차종2_SP2 AT %MW10101.13 : BOOL; (* S362 M 차종2 SP2 *)
    S362_M_차종2_WGN AT %MW10101.11 : BOOL; (* S362 M 차종2 WGN *)
    S362_M_차종3_LHD AT %MW10101.14 : BOOL; (* S362 M 차종3 LHD *)
    S362_M_차종3_RHD AT %MW10101.15 : BOOL; (* S362 M 차종3 RHD *)
    S362_M_차종4_EEC AT %MW10102.3 : BOOL; (* S362 M 차종4 EEC *)
    S362_M_차종4_SP1 AT %MW10102.8 : BOOL; (* S362 M 차종4 SP1 *)
    S362_M_차종4_SP2 AT %MW10102.9 : BOOL; (* S362 M 차종4 SP2 *)
    S362_M_차종4_SP3 AT %MW10102.11 : BOOL; (* S362 M 차종4 SP3 *)
    S362_M_차종4_SP4 AT %MW10102.12 : BOOL; (* S362 M 차종4 SP4 *)
    S362_M_차종4_SP5 AT %MW10102.13 : BOOL; (* S362 M 차종4 SP5 *)
    S362_M_차종4_SP6 AT %MW10102.14 : BOOL; (* S362 M 차종4 SP6 *)
    S362_M_차종4_SP7 AT %MW10102.15 : BOOL; (* S362 M 차종4 SP7 *)
    S362_M_차종4_내수 AT %MW10102.0 : BOOL; (* S362 M 차종4 내수 *)
    S362_M_차종4_러시아 AT %MW10102.10 : BOOL; (* S362 M 차종4 러시아 *)
    S362_M_차종4_북미 AT %MW10102.2 : BOOL; (* S362 M 차종4 북미 *)
    S362_M_차종4_브라질 AT %MW10102.7 : BOOL; (* S362 M 차종4 브라질 *)
    S362_M_차종4_수출 AT %MW10102.1 : BOOL; (* S362 M 차종4 수출 *)
    S362_M_차종4_중국 AT %MW10102.6 : BOOL; (* S362 M 차종4 중국 *)
    S362_M_차종4_중동 AT %MW10102.5 : BOOL; (* S362 M 차종4 중동 *)
    S362_M_차종4_호주 AT %MW10102.4 : BOOL; (* S362 M 차종4 호주 *)
    S362_M_차종5_AT AT %MW10103.1 : BOOL; (* S362 M 차종5 AT *)
    S362_M_차종5_MT AT %MW10103.0 : BOOL; (* S362 M 차종5 MT *)
    S362_M_차종5_SP1 AT %MW10103.2 : BOOL; (* S362 M 차종5 SP1 *)
    S362_M_차종6_DSROOF AT %MW10103.6 : BOOL; (* S362 M 차종6 DSROOF *)
    S362_M_차종6_SP1 AT %MW10103.7 : BOOL; (* S362 M 차종6 SP1 *)
    S362_M_차종6_썬루프 AT %MW10103.4 : BOOL; (* S362 M 차종6 썬루프 *)
    S362_M_차종6_일반루프 AT %MW10103.3 : BOOL; (* S362 M 차종6 일반루프 *)
    S362_M_차종6_파노라마루프 AT %MW10103.5 : BOOL; (* S362 M 차종6 파노라마루프 *)
    S362_M_차종7_DSL AT %MW10103.9 : BOOL; (* S362 M 차종7 DSL *)
    S362_M_차종7_GSL AT %MW10103.8 : BOOL; (* S362 M 차종7 GSL *)
    S362_M_차종7_SP1 AT %MW10103.10 : BOOL; (* S362 M 차종7 SP1 *)
    S362_M_차종7_SP2 AT %MW10103.11 : BOOL; (* S362 M 차종7 SP2 *)
    S362_M_차종7_SP3 AT %MW10103.12 : BOOL; (* S362 M 차종7 SP3 *)
    S362_M_차종7_SP4 AT %MW10103.13 : BOOL; (* S362 M 차종7 SP4 *)
    S362_M_차종7_SP5 AT %MW10103.14 : BOOL; (* S362 M 차종7 SP5 *)
    S362_M_차종7_SP6 AT %MW10103.15 : BOOL; (* S362 M 차종7 SP6 *)
    S362_M_차종8_2WD AT %MW10104.0 : BOOL; (* S362 M 차종8 2WD *)
    S362_M_차종8_4WD AT %MW10104.1 : BOOL; (* S362 M 차종8 4WD *)
    S362_M_차종8_SP1 AT %MW10104.2 : BOOL; (* S362 M 차종8 SP1 *)
    S362_M_차종9_MPI AT %MW10104.3 : BOOL; (* S362 M 차종9 MPI *)
    S362_M_차종9_SP1 AT %MW10104.5 : BOOL; (* S362 M 차종9 SP1 *)
    S362_M_차종9_SP10 AT %MW10104.14 : BOOL; (* S362 M 차종9 SP10 *)
    S362_M_차종9_SP11 AT %MW10104.15 : BOOL; (* S362 M 차종9 SP11 *)
    S362_M_차종9_SP2 AT %MW10104.6 : BOOL; (* S362 M 차종9 SP2 *)
    S362_M_차종9_SP3 AT %MW10104.7 : BOOL; (* S362 M 차종9 SP3 *)
    S362_M_차종9_SP4 AT %MW10104.8 : BOOL; (* S362 M 차종9 SP4 *)
    S362_M_차종9_SP5 AT %MW10104.9 : BOOL; (* S362 M 차종9 SP5 *)
    S362_M_차종9_SP6 AT %MW10104.10 : BOOL; (* S362 M 차종9 SP6 *)
    S362_M_차종9_SP7 AT %MW10104.11 : BOOL; (* S362 M 차종9 SP7 *)
    S362_M_차종9_SP8 AT %MW10104.12 : BOOL; (* S362 M 차종9 SP8 *)
    S362_M_차종9_SP9 AT %MW10104.13 : BOOL; (* S362 M 차종9 SP9 *)
    S362_M_차종9_T_GDI AT %MW10104.4 : BOOL; (* S362 M 차종9 T GDI *)
    S362_M_차종_AS AT %MW10110.9 : BOOL; (* S362 M 차종 AS *)
    S362_M_차종_OPT1_R_RACK_무 AT %MW10105.3 : BOOL; (* S362 M 차종 OPT1 R RACK 무 *)
    S362_M_차종_OPT1_R_RACK_유 AT %MW10105.2 : BOOL; (* S362 M 차종 OPT1 R RACK 유 *)
    S362_M_차종_OPT1_SP1 AT %MW10105.10 : BOOL; (* S362 M 차종 OPT1 SP1 *)
    S362_M_차종_OPT1_SP2 AT %MW10105.11 : BOOL; (* S362 M 차종 OPT1 SP2 *)
    S362_M_차종_OPT1_SP3 AT %MW10105.12 : BOOL; (* S362 M 차종 OPT1 SP3 *)
    S362_M_차종_OPT1_SP4 AT %MW10105.13 : BOOL; (* S362 M 차종 OPT1 SP4 *)
    S362_M_차종_OPT1_SP5 AT %MW10105.14 : BOOL; (* S362 M 차종 OPT1 SP5 *)
    S362_M_차종_OPT1_SP6 AT %MW10105.15 : BOOL; (* S362 M 차종 OPT1 SP6 *)
    S362_M_차종_OPT1_S_REP_EATER_무 AT %MW10105.7 : BOOL; (* S362 M 차종 OPT1 S REP EATER 무 *)
    S362_M_차종_OPT1_S_REP_EATER_유 AT %MW10105.6 : BOOL; (* S362 M 차종 OPT1 S REP EATER 유 *)
    S362_M_차종_OPT1_VAN_무 AT %MW10105.9 : BOOL; (* S362 M 차종 OPT1 VAN 무 *)
    S362_M_차종_OPT1_VAN_유 AT %MW10105.8 : BOOL; (* S362 M 차종 OPT1 VAN 유 *)
    S362_M_차종_OPT1_슬라이딩_무 AT %MW10105.1 : BOOL; (* S362 M 차종 OPT1 슬라이딩 무 *)
    S362_M_차종_OPT1_슬라이딩_유 AT %MW10105.0 : BOOL; (* S362 M 차종 OPT1 슬라이딩 유 *)
    S362_M_차종_OPT1_폴딩_무 AT %MW10105.5 : BOOL; (* S362 M 차종 OPT1 폴딩 무 *)
    S362_M_차종_OPT1_폴딩_유 AT %MW10105.4 : BOOL; (* S362 M 차종 OPT1 폴딩 유 *)
    S362_M_차종_OPT2_SP_WORD1 AT %MW10106 : WORD; (* S362 M 차종 OPT2 SP WORD1 *)
    S362_M_차종_OPT3_SP_WORD2 AT %MW10107 : WORD; (* S362 M 차종 OPT3 SP WORD2 *)
    S362_M_차종_OPT4_SP_WORD3 AT %MW10108 : WORD; (* S362 M 차종 OPT4 SP WORD3 *)
    S362_M_차종_OPT5_SP_WORD4 AT %MW10109 : WORD; (* S362 M 차종 OPT5 SP WORD4 *)
    S362_M_차종_SP1 AT %MW10110.0 : BOOL; (* S362 M 차종 SP1 *)
    S362_M_차종_SP2 AT %MW10110.1 : BOOL; (* S362 M 차종 SP2 *)
    S362_M_차종_SP3 AT %MW10110.2 : BOOL; (* S362 M 차종 SP3 *)
    S362_M_차종_SP4 AT %MW10110.3 : BOOL; (* S362 M 차종 SP4 *)
    S362_M_차종_SP5 AT %MW10110.4 : BOOL; (* S362 M 차종 SP5 *)
    S362_M_차종_SP6 AT %MW10110.5 : BOOL; (* S362 M 차종 SP6 *)
    S362_M_차종_SP7 AT %MW10110.6 : BOOL; (* S362 M 차종 SP7 *)
    S362_M_차종_SP8 AT %MW10110.7 : BOOL; (* S362 M 차종 SP8 *)
    S362_M_차종_SP9 AT %MW10110.15 : BOOL; (* S362 M 차종 SP9 *)
    S362_M_차종_공대차 AT %MW10110.12 : BOOL; (* S362 M 차종 공대차 *)
    S362_M_차종_공차 AT %MW10110.10 : BOOL; (* S362 M 차종 공차 *)
    S362_M_차종_불량대차 AT %MW10110.13 : BOOL; (* S362 M 차종 불량대차 *)
    S362_M_차종_불량차 AT %MW10110.11 : BOOL; (* S362 M 차종 불량차 *)
    S362_M_차종_비축 AT %MW10110.8 : BOOL; (* S362 M 차종 비축 *)
    S362_M_차종_취출대차 AT %MW10110.14 : BOOL; (* S362 M 차종 취출대차 *)
    S362_M_총괄_CP_이상 AT %MW1009.7 : BOOL; (* S362 CP OFF 이상 *)
    S362_M_총괄_CT_이상 AT %MW1010.4 : BOOL; (* S362   TACK TIME 이상 *)
    S362_M_총괄_EOCR_이상 AT %MW1009.8 : BOOL; (* S362_M_총괄_EOCR_이상 *)
    S362_M_총괄_INV_이상 AT %MW1009.9 : BOOL; (* S362 인버터 이상 *)
    S362_M_총괄_LS_이상 AT %MW1009.15 : BOOL; (* S362 LS 이상 *)
    S362_M_총괄_MATCH_이상 AT %MW1010.0 : BOOL; (* S362 매트SW 이상 *)
    S362_M_총괄_MC_이상 AT %MW1009.13 : BOOL; (* S362 MC 이상 *)
    S362_M_총괄_MOTOR_이상 AT %MW1010.3 : BOOL; (* S362 MOTOR 이상 *)
    S362_M_총괄_NFB_이상 AT %MW1009.11 : BOOL; (* S362 NFB 이상 *)
    S362_M_총괄_ROBOT_이상 AT %MW1010.1 : BOOL; (* S362 ROBOT 이상 *)
    S362_M_총괄_SAFETY_이상 AT %MW1009.2 : BOOL; (* S362 SAFETY 이상 *)
    S362_M_총괄_SRV_이상 AT %MW1009.10 : BOOL; (* S362_M_총괄_SRV_이상 *)
    S362_M_총괄_공기압_이상 AT %MW1009.3 : BOOL; (* S362 공기압 이상 *)
    S362_M_총괄_비상정지_이상 AT %MW1009.1 : BOOL; (* S362_M_총괄_비상정지_이상 *)
    S362_M_총괄_사양_이상 AT %MW1009.6 : BOOL; (* S362 사양 이상 *)
    S362_M_총괄_오버런_이상 AT %MW1009.12 : BOOL; (* S362 OVER RUN 이상 *)
    S362_M_총괄_용접타점수_이상 AT %MW1010.2 : BOOL; (* S362 용접타점수 이상 *)
    S362_M_총괄_이상 AT %MW1009.0 : BOOL; (* S362_M_총괄_이상 *)
    S362_M_총괄_제품감지_이상 AT %MW1009.4 : BOOL; (* S362 제품감지 이상 *)
    S362_M_총괄_차종_이상 AT %MW1009.5 : BOOL; (* S362 차종 이상 *)
    S362_M_총괄_통신_이상 AT %MW1009.14 : BOOL; (* S362 통신이상 *)
    S362_전진_ON AT %MW1048.1 : BOOL; (* S362_전진_ON *)
    S362_후진_ON AT %MW1048.2 : BOOL; (* S362_후진_ON *)
    S364_HOME AT %MW2048.0 : BOOL; (* S364_HOME *)
    S364_LH_M_NODE_7_16_통신_이상 AT %MW2024.0 : BOOL;
    S364_M_AOP_비상정지_이상 AT %MW2011.0 : BOOL; (* S364_M_AOP_비상정지_이상 *)
    S364_M_AX_CLAMP_전진_LS_이상 AT %MW2101.5 : BOOL; (* S364_M_AX_CLAMP_전진_LS_이상 *)
    S364_M_AX_CLAMP_전진_보조 AT %MW2101.1 : BOOL; (* S364_M_AX_CLAMP_전진_보조 *)
    S364_M_AX_CLAMP_전진단 AT %MW2101.3 : BOOL; (* S364_M_AX_CLAMP_전진단 *)
    S364_M_AX_CLAMP_조건 AT %MW2101.0 : BOOL; (* S364_M_AX_CLAMP_조건 *)
    S364_M_AX_CLAMP_후진_LS_이상 AT %MW2101.6 : BOOL; (* S364_M_AX_CLAMP_후진_LS_이상 *)
    S364_M_AX_CLAMP_후진_보조 AT %MW2101.2 : BOOL; (* S364_M_AX_CLAMP_후진_보조 *)
    S364_M_AX_CLAMP_후진단 AT %MW2101.4 : BOOL; (* S364_M_AX_CLAMP_후진단 *)
    S364_M_AX_LATCH_전진_LS_이상 AT %MW2100.5 : BOOL; (* S364_M_AX_LATCH_전진_LS_이상 *)
    S364_M_AX_LATCH_전진_보조 AT %MW2100.1 : BOOL; (* S364_M_AX_LATCH_전진_보조 *)
    S364_M_AX_LATCH_전진단 AT %MW2100.3 : BOOL; (* S364_M_AX_LATCH_전진단 *)
    S364_M_AX_LATCH_조건 AT %MW2100.0 : BOOL; (* S364_M_AX_LATCH_조건 *)
    S364_M_AX_LATCH_후진_LS_이상 AT %MW2100.6 : BOOL; (* S364_M_AX_LATCH_후진_LS_이상 *)
    S364_M_AX_LATCH_후진_보조 AT %MW2100.2 : BOOL; (* S364_M_AX_LATCH_후진_보조 *)
    S364_M_AX_LATCH_후진단 AT %MW2100.4 : BOOL; (* S364_M_AX_LATCH_후진단 *)
    S364_M_AX_LH_SLD_CLP_전진_LS_이상 AT %MW2103.5 : BOOL; (* S364_M_AX_LH_SLD_CLP_전진_LS_이상 *)
    S364_M_AX_LH_SLD_CLP_전진_보조 AT %MW2103.1 : BOOL; (* S364_M_AX_LH_SLD_CLP_전진_보조 *)
    S364_M_AX_LH_SLD_CLP_전진단 AT %MW2103.3 : BOOL; (* S364_M_AX_LH_SLD_CLP_전진단 *)
    S364_M_AX_LH_SLD_CLP_조건 AT %MW2103.0 : BOOL; (* S364_M_AX_LH_SLD_CLP_조건 *)
    S364_M_AX_LH_SLD_CLP_후진_LS_이상 AT %MW2103.6 : BOOL; (* S364_M_AX_LH_SLD_CLP_후진_LS_이상 *)
    S364_M_AX_LH_SLD_CLP_후진_보조 AT %MW2103.2 : BOOL; (* S364_M_AX_LH_SLD_CLP_후진_보조 *)
    S364_M_AX_LH_SLD_CLP_후진단 AT %MW2103.4 : BOOL; (* S364_M_AX_LH_SLD_CLP_후진단 *)
    S364_M_AX_LH_SLD_LAT_전진_LS_이상 AT %MW2102.5 : BOOL; (* S364_M_AX_LH_SLD_LAT_전진_LS_이상 *)
    S364_M_AX_LH_SLD_LAT_전진_보조 AT %MW2102.1 : BOOL; (* S364_M_AX_LH_SLD_LAT_전진_보조 *)
    S364_M_AX_LH_SLD_LAT_전진단 AT %MW2102.3 : BOOL; (* S364_M_AX_LH_SLD_LAT_전진단 *)
    S364_M_AX_LH_SLD_LAT_조건 AT %MW2102.0 : BOOL; (* S364_M_AX_LH_SLD_LAT_조건 *)
    S364_M_AX_LH_SLD_LAT_후진_LS_이상 AT %MW2102.6 : BOOL; (* S364_M_AX_LH_SLD_LAT_후진_LS_이상 *)
    S364_M_AX_LH_SLD_LAT_후진_보조 AT %MW2102.2 : BOOL; (* S364_M_AX_LH_SLD_LAT_후진_보조 *)
    S364_M_AX_LH_SLD_LAT_후진단 AT %MW2102.4 : BOOL; (* S364_M_AX_LH_SLD_LAT_후진단 *)
    S364_M_AX_LH_SLD_전진_LS_이상 AT %MW2107.5 : BOOL; (* S364_M_AX_LH_SLD_전진_LS_이상 *)
    S364_M_AX_LH_SLD_전진_보조 AT %MW2107.1 : BOOL; (* S364_M_AX_LH_SLD_전진_보조 *)
    S364_M_AX_LH_SLD_전진단 AT %MW2107.3 : BOOL; (* S364_M_AX_LH_SLD_전진단 *)
    S364_M_AX_LH_SLD_조건 AT %MW2107.0 : BOOL; (* S364_M_AX_LH_SLD_조건 *)
    S364_M_AX_LH_SLD_후진_LS_이상 AT %MW2107.6 : BOOL; (* S364_M_AX_LH_SLD_후진_LS_이상 *)
    S364_M_AX_LH_SLD_후진_보조 AT %MW2107.2 : BOOL; (* S364_M_AX_LH_SLD_후진_보조 *)
    S364_M_AX_LH_SLD_후진단 AT %MW2107.4 : BOOL; (* S364_M_AX_LH_SLD_후진단 *)
    S364_M_AX_RH_SLD_CLP_전진_LS_이상 AT %MW2111.5 : BOOL; (* S364_M_AX_RH_SLD_CLP_전진_LS_이상 *)
    S364_M_AX_RH_SLD_CLP_전진_보조 AT %MW2111.1 : BOOL; (* S364_M_AX_RH_SLD_CLP_전진_보조 *)
    S364_M_AX_RH_SLD_CLP_전진단 AT %MW2111.3 : BOOL; (* S364_M_AX_RH_SLD_CLP_전진단 *)
    S364_M_AX_RH_SLD_CLP_조건 AT %MW2111.0 : BOOL; (* S364_M_AX_RH_SLD_CLP_조건 *)
    S364_M_AX_RH_SLD_CLP_후진_LS_이상 AT %MW2111.6 : BOOL; (* S364_M_AX_RH_SLD_CLP_후진_LS_이상 *)
    S364_M_AX_RH_SLD_CLP_후진_보조 AT %MW2111.2 : BOOL; (* S364_M_AX_RH_SLD_CLP_후진_보조 *)
    S364_M_AX_RH_SLD_CLP_후진단 AT %MW2111.4 : BOOL; (* S364_M_AX_RH_SLD_CLP_후진단 *)
    S364_M_AX_RH_SLD_LAT_전진_LS_이상 AT %MW2110.5 : BOOL; (* S364_M_AX_RH_SLD_LAT_전진_LS_이상 *)
    S364_M_AX_RH_SLD_LAT_전진_보조 AT %MW2110.1 : BOOL; (* S364_M_AX_RH_SLD_LAT_전진_보조 *)
    S364_M_AX_RH_SLD_LAT_전진단 AT %MW2110.3 : BOOL; (* S364_M_AX_RH_SLD_LAT_전진단 *)
    S364_M_AX_RH_SLD_LAT_조건 AT %MW2110.0 : BOOL; (* S364_M_AX_RH_SLD_LAT_조건 *)
    S364_M_AX_RH_SLD_LAT_후진_LS_이상 AT %MW2110.6 : BOOL; (* S364_M_AX_RH_SLD_LAT_후진_LS_이상 *)
    S364_M_AX_RH_SLD_LAT_후진_보조 AT %MW2110.2 : BOOL; (* S364_M_AX_RH_SLD_LAT_후진_보조 *)
    S364_M_AX_RH_SLD_LAT_후진단 AT %MW2110.4 : BOOL; (* S364_M_AX_RH_SLD_LAT_후진단 *)
    S364_M_AX_RH_SLD_전진_LS_이상 AT %MW2115.5 : BOOL; (* S364_M_AX_RH_SLD_전진_LS_이상 *)
    S364_M_AX_RH_SLD_전진_보조 AT %MW2115.1 : BOOL; (* S364_M_AX_RH_SLD_전진_보조 *)
    S364_M_AX_RH_SLD_전진단 AT %MW2115.3 : BOOL; (* S364_M_AX_RH_SLD_전진단 *)
    S364_M_AX_RH_SLD_조건 AT %MW2115.0 : BOOL; (* S364_M_AX_RH_SLD_조건 *)
    S364_M_AX_RH_SLD_후진_LS_이상 AT %MW2115.6 : BOOL; (* S364_M_AX_RH_SLD_후진_LS_이상 *)
    S364_M_AX_RH_SLD_후진_보조 AT %MW2115.2 : BOOL; (* S364_M_AX_RH_SLD_후진_보조 *)
    S364_M_AX_RH_SLD_후진단 AT %MW2115.4 : BOOL; (* S364_M_AX_RH_SLD_후진단 *)
    S364_M_BYPASS_보조 AT %MW2003.15 : BOOL; (* S364 M BYPASS 보조 *)
    S364_M_CTIME_OVER_ALRAM AT %MW2007.14 : BOOL; (* S364_M_CTIME_OVER_ALRAM *)
    S364_M_CTIME_OVER_MUTE AT %MW2007.13 : BOOL; (* S364_M_CTIME_OVER_MUTE *)
    S364_M_CTR_RACK_제품감지_무 AT %MW2002.9 : BOOL;
    S364_M_CTR_RACK_제품감지_유 AT %MW2002.8 : BOOL;
    S364_M_CTR_RACK_제품감지_이상 AT %MW2014.1 : BOOL;
    S364_M_DATA_삭제_PLS AT %MW9012.0 : BOOL; (* S364 M DATA 삭제 PLS *)
    S364_M_DATA_삭제_SIGN AT %MW9012.1 : BOOL; (* S364 M DATA 삭제 SIGN *)
    S364_M_DATA_삭제_완료 AT %MW9012.2 : BOOL; (* S364 M DATA 삭제 완료 *)
    S364_M_FRT_PNL_제품감지_무 AT %MW2002.13 : BOOL;
